	        ELSIF (#i_UDT_PDPStatus.Specific.CircuitBreakerTrippedF108 <> #s_UDT_PDPOldStatus.Specific.CircuitBreakerTrippedF108 AND NOT #sx_SendAllProcedure)
	            OR (#sx_SendAllProcedure AND #ii_ErrorNumber = 10)
	        THEN
	            #sdi_Code := "DB_MFC_ErrorCode".PDP.CircuitBreakerTrippedF108;
	            #si_State := BOOL_TO_INT(#i_UDT_PDPStatus.Specific.CircuitBreakerTrippedF108);
	            #s_UDT_PDPOldStatus.Specific.CircuitBreakerTrippedF108 := #i_UDT_PDPStatus.Specific.CircuitBreakerTrippedF108;
	            #sx_ItemErrorMessageReq := TRUE;
	            #ii_ErrorNumber += 1;
	        ELSIF (#i_UDT_PDPStatus.Specific.CircuitBreakerTrippedF109 <> #s_UDT_PDPOldStatus.Specific.CircuitBreakerTrippedF109 AND NOT #sx_SendAllProcedure)
	            OR (#sx_SendAllProcedure AND #ii_ErrorNumber = 11)
	        THEN
	            #sdi_Code := "DB_MFC_ErrorCode".PDP.CircuitBreakerTrippedF109;
	            #si_State := BOOL_TO_INT(#i_UDT_PDPStatus.Specific.CircuitBreakerTrippedF109);
	            #s_UDT_PDPOldStatus.Specific.CircuitBreakerTrippedF109 := #i_UDT_PDPStatus.Specific.CircuitBreakerTrippedF109;
	            #sx_ItemErrorMessageReq := TRUE;
	            #ii_ErrorNumber += 1;
	        ELSIF (#i_UDT_PDPStatus.Specific.CircuitBreakerTrippedF110 <> #s_UDT_PDPOldStatus.Specific.CircuitBreakerTrippedF110 AND NOT #sx_SendAllProcedure)
	            OR (#sx_SendAllProcedure AND #ii_ErrorNumber = 12)
	        THEN
	            #sdi_Code := "DB_MFC_ErrorCode".PDP.CircuitBreakerTrippedF110;
	            #si_State := BOOL_TO_INT(#i_UDT_PDPStatus.Specific.CircuitBreakerTrippedF110);
	            #s_UDT_PDPOldStatus.Specific.CircuitBreakerTrippedF110 := #i_UDT_PDPStatus.Specific.CircuitBreakerTrippedF110;
	            #sx_ItemErrorMessageReq := TRUE;
	            #ii_ErrorNumber += 1;
	        ELSIF (#i_UDT_PDPStatus.Specific.CircuitBreakerTrippedF111 <> #s_UDT_PDPOldStatus.Specific.CircuitBreakerTrippedF111 AND NOT #sx_SendAllProcedure)
	            OR (#sx_SendAllProcedure AND #ii_ErrorNumber = 13)
	        THEN
	            #sdi_Code := "DB_MFC_ErrorCode".PDP.CircuitBreakerTrippedF111;
	            #si_State := BOOL_TO_INT(#i_UDT_PDPStatus.Specific.CircuitBreakerTrippedF111);
	            #s_UDT_PDPOldStatus.Specific.CircuitBreakerTrippedF111 := #i_UDT_PDPStatus.Specific.CircuitBreakerTrippedF111;
	            #sx_ItemErrorMessageReq := TRUE;
	            #ii_ErrorNumber += 1;
	        ELSIF (#i_UDT_PDPStatus.Specific.CircuitBreakerTrippedF112 <> #s_UDT_PDPOldStatus.Specific.CircuitBreakerTrippedF112 AND NOT #sx_SendAllProcedure)
	            OR (#sx_SendAllProcedure AND #ii_ErrorNumber = 14)
	        THEN
	            #sdi_Code := "DB_MFC_ErrorCode".PDP.CircuitBreakerTrippedF112;
	            #si_State := BOOL_TO_INT(#i_UDT_PDPStatus.Specific.CircuitBreakerTrippedF112);
	            #s_UDT_PDPOldStatus.Specific.CircuitBreakerTrippedF112 := #i_UDT_PDPStatus.Specific.CircuitBreakerTrippedF112;
	            #sx_ItemErrorMessageReq := TRUE;
	            #ii_ErrorNumber += 1;
	        ELSIF (#i_UDT_PDPStatus.Specific.CircuitBreakerTrippedF113 <> #s_UDT_PDPOldStatus.Specific.CircuitBreakerTrippedF113 AND NOT #sx_SendAllProcedure)
	            OR (#sx_SendAllProcedure AND #ii_ErrorNumber = 15)
	        THEN
	            #sdi_Code := "DB_MFC_ErrorCode".PDP.CircuitBreakerTrippedF113;
	            #si_State := BOOL_TO_INT(#i_UDT_PDPStatus.Specific.CircuitBreakerTrippedF113);
	            #s_UDT_PDPOldStatus.Specific.CircuitBreakerTrippedF113 := #i_UDT_PDPStatus.Specific.CircuitBreakerTrippedF113;
	            #sx_ItemErrorMessageReq := TRUE;
	            #ii_ErrorNumber += 1;
	        ELSIF (#i_UDT_PDPStatus.Specific.CircuitBreakerTrippedF114 <> #s_UDT_PDPOldStatus.Specific.CircuitBreakerTrippedF114 AND NOT #sx_SendAllProcedure)
	            OR (#sx_SendAllProcedure AND #ii_ErrorNumber = 16)
	        THEN
	            #sdi_Code := "DB_MFC_ErrorCode".PDP.CircuitBreakerTrippedF114;
	            #si_State := BOOL_TO_INT(#i_UDT_PDPStatus.Specific.CircuitBreakerTrippedF114);
	            #s_UDT_PDPOldStatus.Specific.CircuitBreakerTrippedF114 := #i_UDT_PDPStatus.Specific.CircuitBreakerTrippedF114;
	            #sx_ItemErrorMessageReq := TRUE;
	            #ii_ErrorNumber += 1;
	        ELSIF (#i_UDT_PDPStatus.Specific.CircuitBreakerTrippedF115 <> #s_UDT_PDPOldStatus.Specific.CircuitBreakerTrippedF115 AND NOT #sx_SendAllProcedure)
	            OR (#sx_SendAllProcedure AND #ii_ErrorNumber = 17)
	        THEN
	            #sdi_Code := "DB_MFC_ErrorCode".PDP.CircuitBreakerTrippedF115;
	            #si_State := BOOL_TO_INT(#i_UDT_PDPStatus.Specific.CircuitBreakerTrippedF115);
	            #s_UDT_PDPOldStatus.Specific.CircuitBreakerTrippedF115 := #i_UDT_PDPStatus.Specific.CircuitBreakerTrippedF115;
	            #sx_ItemErrorMessageReq := TRUE;
	            #ii_ErrorNumber += 1;
	        ELSIF (#i_UDT_PDPStatus.Specific.CircuitBreakerTrippedF116 <> #s_UDT_PDPOldStatus.Specific.CircuitBreakerTrippedF116 AND NOT #sx_SendAllProcedure)
	            OR (#sx_SendAllProcedure AND #ii_ErrorNumber = 18)
	        THEN
	            #sdi_Code := "DB_MFC_ErrorCode".PDP.CircuitBreakerTrippedF116;
	            #si_State := BOOL_TO_INT(#i_UDT_PDPStatus.Specific.CircuitBreakerTrippedF116);
	            #s_UDT_PDPOldStatus.Specific.CircuitBreakerTrippedF116 := #i_UDT_PDPStatus.Specific.CircuitBreakerTrippedF116;
	            #sx_ItemErrorMessageReq := TRUE;
	            #ii_ErrorNumber += 1;
	        ELSIF (#i_UDT_PDPStatus.Specific.CircuitBreakerTrippedF117 <> #s_UDT_PDPOldStatus.Specific.CircuitBreakerTrippedF117 AND NOT #sx_SendAllProcedure)
	            OR (#sx_SendAllProcedure AND #ii_ErrorNumber = 19)
	        THEN
	            #sdi_Code := "DB_MFC_ErrorCode".PDP.CircuitBreakerTrippedF117;
	            #si_State := BOOL_TO_INT(#i_UDT_PDPStatus.Specific.CircuitBreakerTrippedF117);
	            #s_UDT_PDPOldStatus.Specific.CircuitBreakerTrippedF117 := #i_UDT_PDPStatus.Specific.CircuitBreakerTrippedF117;
	            #sx_ItemErrorMessageReq := TRUE;
	            #ii_ErrorNumber += 1;
	        ELSIF (#i_UDT_PDPStatus.Specific.CircuitBreakerTrippedF118 <> #s_UDT_PDPOldStatus.Specific.CircuitBreakerTrippedF118 AND NOT #sx_SendAllProcedure)
	            OR (#sx_SendAllProcedure AND #ii_ErrorNumber = 20)
	        THEN
	            #sdi_Code := "DB_MFC_ErrorCode".PDP.CircuitBreakerTrippedF118;
	            #si_State := BOOL_TO_INT(#i_UDT_PDPStatus.Specific.CircuitBreakerTrippedF118);
	            #s_UDT_PDPOldStatus.Specific.CircuitBreakerTrippedF118 := #i_UDT_PDPStatus.Specific.CircuitBreakerTrippedF118;
	            #sx_ItemErrorMessageReq := TRUE;
	            #ii_ErrorNumber += 1;
	        ELSIF (#i_UDT_PDPStatus.Specific.CircuitBreakerTrippedF119 <> #s_UDT_PDPOldStatus.Specific.CircuitBreakerTrippedF119 AND NOT #sx_SendAllProcedure)
	            OR (#sx_SendAllProcedure AND #ii_ErrorNumber = 21)
	        THEN
	            #sdi_Code := "DB_MFC_ErrorCode".PDP.CircuitBreakerTrippedF119;
	            #si_State := BOOL_TO_INT(#i_UDT_PDPStatus.Specific.CircuitBreakerTrippedF119);
	            #s_UDT_PDPOldStatus.Specific.CircuitBreakerTrippedF119 := #i_UDT_PDPStatus.Specific.CircuitBreakerTrippedF119;
	            #sx_ItemErrorMessageReq := TRUE;
	            #ii_ErrorNumber += 1;
	        ELSIF (#i_UDT_PDPStatus.Specific.CircuitBreakerTrippedF120 <> #s_UDT_PDPOldStatus.Specific.CircuitBreakerTrippedF120 AND NOT #sx_SendAllProcedure)
	            OR (#sx_SendAllProcedure AND #ii_ErrorNumber = 22)
	        THEN
	            #sdi_Code := "DB_MFC_ErrorCode".PDP.CircuitBreakerTrippedF120;
	            #si_State := BOOL_TO_INT(#i_UDT_PDPStatus.Specific.CircuitBreakerTrippedF120);
	            #s_UDT_PDPOldStatus.Specific.CircuitBreakerTrippedF120 := #i_UDT_PDPStatus.Specific.CircuitBreakerTrippedF120;
	            #sx_ItemErrorMessageReq := TRUE;
	            #ii_ErrorNumber += 1;
	        ELSIF (#i_UDT_PDPStatus.Specific.CircuitBreakerTrippedF121 <> #s_UDT_PDPOldStatus.Specific.CircuitBreakerTrippedF121 AND NOT #sx_SendAllProcedure)
	            OR (#sx_SendAllProcedure AND #ii_ErrorNumber = 23)
	        THEN
	            #sdi_Code := "DB_MFC_ErrorCode".PDP.CircuitBreakerTrippedF121;
	            #si_State := BOOL_TO_INT(#i_UDT_PDPStatus.Specific.CircuitBreakerTrippedF121);
	            #s_UDT_PDPOldStatus.Specific.CircuitBreakerTrippedF121 := #i_UDT_PDPStatus.Specific.CircuitBreakerTrippedF121;
	            #sx_ItemErrorMessageReq := TRUE;
	            #ii_ErrorNumber += 1;
	        ELSIF (#i_UDT_PDPStatus.Specific.CircuitBreakerTrippedF122 <> #s_UDT_PDPOldStatus.Specific.CircuitBreakerTrippedF122 AND NOT #sx_SendAllProcedure)
	            OR (#sx_SendAllProcedure AND #ii_ErrorNumber = 24)
	        THEN
	            #sdi_Code := "DB_MFC_ErrorCode".PDP.CircuitBreakerTrippedF122;
	            #si_State := BOOL_TO_INT(#i_UDT_PDPStatus.Specific.CircuitBreakerTrippedF122);
	            #s_UDT_PDPOldStatus.Specific.CircuitBreakerTrippedF122 := #i_UDT_PDPStatus.Specific.CircuitBreakerTrippedF122;
	            #sx_ItemErrorMessageReq := TRUE;
	            #ii_ErrorNumber += 1;
	        ELSIF (#i_UDT_PDPStatus.Specific.CircuitBreakerTrippedF123 <> #s_UDT_PDPOldStatus.Specific.CircuitBreakerTrippedF123 AND NOT #sx_SendAllProcedure)
	            OR (#sx_SendAllProcedure AND #ii_ErrorNumber = 25)
	        THEN
	            #sdi_Code := "DB_MFC_ErrorCode".PDP.CircuitBreakerTrippedF123;
	            #si_State := BOOL_TO_INT(#i_UDT_PDPStatus.Specific.CircuitBreakerTrippedF123);
	            #s_UDT_PDPOldStatus.Specific.CircuitBreakerTrippedF123 := #i_UDT_PDPStatus.Specific.CircuitBreakerTrippedF123;
	            #sx_ItemErrorMessageReq := TRUE;
	            #ii_ErrorNumber += 1;
	        ELSIF (#i_UDT_PDPStatus.Specific.CircuitBreakerTrippedF124 <> #s_UDT_PDPOldStatus.Specific.CircuitBreakerTrippedF124 AND NOT #sx_SendAllProcedure)
	            OR (#sx_SendAllProcedure AND #ii_ErrorNumber = 26)
	        THEN
	            #sdi_Code := "DB_MFC_ErrorCode".PDP.CircuitBreakerTrippedF124;
	            #si_State := BOOL_TO_INT(#i_UDT_PDPStatus.Specific.CircuitBreakerTrippedF124);
	            #s_UDT_PDPOldStatus.Specific.CircuitBreakerTrippedF124 := #i_UDT_PDPStatus.Specific.CircuitBreakerTrippedF124;
	            #sx_ItemErrorMessageReq := TRUE;
	            #ii_ErrorNumber += 1;
	        ELSIF (#i_UDT_PDPStatus.Specific.CircuitBreakerTrippedF125 <> #s_UDT_PDPOldStatus.Specific.CircuitBreakerTrippedF125 AND NOT #sx_SendAllProcedure)
	            OR (#sx_SendAllProcedure AND #ii_ErrorNumber = 27)
	        THEN
	            #sdi_Code := "DB_MFC_ErrorCode".PDP.CircuitBreakerTrippedF125;
	            #si_State := BOOL_TO_INT(#i_UDT_PDPStatus.Specific.CircuitBreakerTrippedF125);
	            #s_UDT_PDPOldStatus.Specific.CircuitBreakerTrippedF125 := #i_UDT_PDPStatus.Specific.CircuitBreakerTrippedF125;
	            #sx_ItemErrorMessageReq := TRUE;
	            #ii_ErrorNumber += 1;
	        ELSIF (#i_UDT_PDPStatus.Specific.CircuitBreakerTrippedF126 <> #s_UDT_PDPOldStatus.Specific.CircuitBreakerTrippedF126 AND NOT #sx_SendAllProcedure)
	            OR (#sx_SendAllProcedure AND #ii_ErrorNumber = 28)
	        THEN
	            #sdi_Code := "DB_MFC_ErrorCode".PDP.CircuitBreakerTrippedF126;
	            #si_State := BOOL_TO_INT(#i_UDT_PDPStatus.Specific.CircuitBreakerTrippedF126);
	            #s_UDT_PDPOldStatus.Specific.CircuitBreakerTrippedF126 := #i_UDT_PDPStatus.Specific.CircuitBreakerTrippedF126;
	            #sx_ItemErrorMessageReq := TRUE;
	            #ii_ErrorNumber += 1;
	        ELSIF (#i_UDT_PDPStatus.Specific.CircuitBreakerTrippedF127 <> #s_UDT_PDPOldStatus.Specific.CircuitBreakerTrippedF127 AND NOT #sx_SendAllProcedure)
	            OR (#sx_SendAllProcedure AND #ii_ErrorNumber = 29)
	        THEN
	            #sdi_Code := "DB_MFC_ErrorCode".PDP.CircuitBreakerTrippedF127;
	            #si_State := BOOL_TO_INT(#i_UDT_PDPStatus.Specific.CircuitBreakerTrippedF127);
	            #s_UDT_PDPOldStatus.Specific.CircuitBreakerTrippedF127 := #i_UDT_PDPStatus.Specific.CircuitBreakerTrippedF127;
	            #sx_ItemErrorMessageReq := TRUE;
	            #ii_ErrorNumber += 1;
	        ELSIF (#i_UDT_PDPStatus.Specific.CircuitBreakerTrippedF128 <> #s_UDT_PDPOldStatus.Specific.CircuitBreakerTrippedF128 AND NOT #sx_SendAllProcedure)
	            OR (#sx_SendAllProcedure AND #ii_ErrorNumber = 30)
	        THEN
	            #sdi_Code := "DB_MFC_ErrorCode".PDP.CircuitBreakerTrippedF128;
	            #si_State := BOOL_TO_INT(#i_UDT_PDPStatus.Specific.CircuitBreakerTrippedF128);
	            #s_UDT_PDPOldStatus.Specific.CircuitBreakerTrippedF128 := #i_UDT_PDPStatus.Specific.CircuitBreakerTrippedF128;
	            #sx_ItemErrorMessageReq := TRUE;
	            #ii_ErrorNumber += 1;
	        ELSIF (#i_UDT_PDPStatus.Specific.CircuitBreakerTrippedF129 <> #s_UDT_PDPOldStatus.Specific.CircuitBreakerTrippedF129 AND NOT #sx_SendAllProcedure)
	            OR (#sx_SendAllProcedure AND #ii_ErrorNumber = 31)
	        THEN
	            #sdi_Code := "DB_MFC_ErrorCode".PDP.CircuitBreakerTrippedF129;
	            #si_State := BOOL_TO_INT(#i_UDT_PDPStatus.Specific.CircuitBreakerTrippedF129);
	            #s_UDT_PDPOldStatus.Specific.CircuitBreakerTrippedF129 := #i_UDT_PDPStatus.Specific.CircuitBreakerTrippedF129;
	            #sx_ItemErrorMessageReq := TRUE;
	            #ii_ErrorNumber += 1;
	        ELSIF (#i_UDT_PDPStatus.Specific.CircuitBreakerTrippedF130 <> #s_UDT_PDPOldStatus.Specific.CircuitBreakerTrippedF130 AND NOT #sx_SendAllProcedure)
	            OR (#sx_SendAllProcedure AND #ii_ErrorNumber = 32)
	        THEN
	            #sdi_Code := "DB_MFC_ErrorCode".PDP.CircuitBreakerTrippedF130;
	            #si_State := BOOL_TO_INT(#i_UDT_PDPStatus.Specific.CircuitBreakerTrippedF130);
	            #s_UDT_PDPOldStatus.Specific.CircuitBreakerTrippedF130 := #i_UDT_PDPStatus.Specific.CircuitBreakerTrippedF130;
	            #sx_ItemErrorMessageReq := TRUE;
	            #ii_ErrorNumber += 1;
	        ELSIF (#i_UDT_PDPStatus.Specific.CircuitBreakerTrippedF131 <> #s_UDT_PDPOldStatus.Specific.CircuitBreakerTrippedF131 AND NOT #sx_SendAllProcedure)
	            OR (#sx_SendAllProcedure AND #ii_ErrorNumber = 33)
	        THEN
	            #sdi_Code := "DB_MFC_ErrorCode".PDP.CircuitBreakerTrippedF131;
	            #si_State := BOOL_TO_INT(#i_UDT_PDPStatus.Specific.CircuitBreakerTrippedF131);
	            #s_UDT_PDPOldStatus.Specific.CircuitBreakerTrippedF131 := #i_UDT_PDPStatus.Specific.CircuitBreakerTrippedF131;
	            #sx_ItemErrorMessageReq := TRUE;
	            #ii_ErrorNumber += 1;
	        ELSIF (#i_UDT_PDPStatus.Specific.CircuitBreakerTrippedF132 <> #s_UDT_PDPOldStatus.Specific.CircuitBreakerTrippedF132 AND NOT #sx_SendAllProcedure)
	            OR (#sx_SendAllProcedure AND #ii_ErrorNumber = 34)
	        THEN
	            #sdi_Code := "DB_MFC_ErrorCode".PDP.CircuitBreakerTrippedF132;
	            #si_State := BOOL_TO_INT(#i_UDT_PDPStatus.Specific.CircuitBreakerTrippedF132);
	            #s_UDT_PDPOldStatus.Specific.CircuitBreakerTrippedF132 := #i_UDT_PDPStatus.Specific.CircuitBreakerTrippedF132;
	            #sx_ItemErrorMessageReq := TRUE;
	            #ii_ErrorNumber += 1;
	        ELSIF (#i_UDT_PDPStatus.Specific.CircuitBreakerTrippedF133 <> #s_UDT_PDPOldStatus.Specific.CircuitBreakerTrippedF133 AND NOT #sx_SendAllProcedure)
	            OR (#sx_SendAllProcedure AND #ii_ErrorNumber = 35)
	        THEN
	            #sdi_Code := "DB_MFC_ErrorCode".PDP.CircuitBreakerTrippedF133;
	            #si_State := BOOL_TO_INT(#i_UDT_PDPStatus.Specific.CircuitBreakerTrippedF133);
	            #s_UDT_PDPOldStatus.Specific.CircuitBreakerTrippedF133 := #i_UDT_PDPStatus.Specific.CircuitBreakerTrippedF133;
	            #sx_ItemErrorMessageReq := TRUE;
	            #ii_ErrorNumber += 1;
	        ELSIF (#i_UDT_PDPStatus.Specific.CircuitBreakerTrippedF134 <> #s_UDT_PDPOldStatus.Specific.CircuitBreakerTrippedF134 AND NOT #sx_SendAllProcedure)
	            OR (#sx_SendAllProcedure AND #ii_ErrorNumber = 36)
	        THEN
	            #sdi_Code := "DB_MFC_ErrorCode".PDP.CircuitBreakerTrippedF134;
	            #si_State := BOOL_TO_INT(#i_UDT_PDPStatus.Specific.CircuitBreakerTrippedF134);
	            #s_UDT_PDPOldStatus.Specific.CircuitBreakerTrippedF134 := #i_UDT_PDPStatus.Specific.CircuitBreakerTrippedF134;
	            #sx_ItemErrorMessageReq := TRUE;
	            #ii_ErrorNumber += 1;
	        ELSIF (#i_UDT_PDPStatus.Specific.CircuitBreakerTrippedF135 <> #s_UDT_PDPOldStatus.Specific.CircuitBreakerTrippedF135 AND NOT #sx_SendAllProcedure)
	            OR (#sx_SendAllProcedure AND #ii_ErrorNumber = 37)
	        THEN
	            #sdi_Code := "DB_MFC_ErrorCode".PDP.CircuitBreakerTrippedF135;
	            #si_State := BOOL_TO_INT(#i_UDT_PDPStatus.Specific.CircuitBreakerTrippedF135);
	            #s_UDT_PDPOldStatus.Specific.CircuitBreakerTrippedF135 := #i_UDT_PDPStatus.Specific.CircuitBreakerTrippedF135;
	            #sx_ItemErrorMessageReq := TRUE;
	            #ii_ErrorNumber += 1;
	        ELSIF (#i_UDT_PDPStatus.Specific.CircuitBreakerTrippedF201 <> #s_UDT_PDPOldStatus.Specific.CircuitBreakerTrippedF201 AND NOT #sx_SendAllProcedure)
	            OR (#sx_SendAllProcedure AND #ii_ErrorNumber = 38)
	        THEN
	            #sdi_Code := "DB_MFC_ErrorCode".PDP.CircuitBreakerTrippedF201;
	            #si_State := BOOL_TO_INT(#i_UDT_PDPStatus.Specific.CircuitBreakerTrippedF201);
	            #s_UDT_PDPOldStatus.Specific.CircuitBreakerTrippedF201 := #i_UDT_PDPStatus.Specific.CircuitBreakerTrippedF201;
	            #sx_ItemErrorMessageReq := TRUE;
	            #ii_ErrorNumber += 1;
	        ELSIF (#i_UDT_PDPStatus.Specific.CircuitBreakerTrippedF202 <> #s_UDT_PDPOldStatus.Specific.CircuitBreakerTrippedF202 AND NOT #sx_SendAllProcedure)
	            OR (#sx_SendAllProcedure AND #ii_ErrorNumber = 39)
	        THEN
	            #sdi_Code := "DB_MFC_ErrorCode".PDP.CircuitBreakerTrippedF202;
	            #si_State := BOOL_TO_INT(#i_UDT_PDPStatus.Specific.CircuitBreakerTrippedF202);
	            #s_UDT_PDPOldStatus.Specific.CircuitBreakerTrippedF202 := #i_UDT_PDPStatus.Specific.CircuitBreakerTrippedF202;
	            #sx_ItemErrorMessageReq := TRUE;
	            #ii_ErrorNumber += 1;
	        ELSIF (#i_UDT_PDPStatus.Specific.CircuitBreakerTrippedF203 <> #s_UDT_PDPOldStatus.Specific.CircuitBreakerTrippedF203 AND NOT #sx_SendAllProcedure)
	            OR (#sx_SendAllProcedure AND #ii_ErrorNumber = 40)
	        THEN
	            #sdi_Code := "DB_MFC_ErrorCode".PDP.CircuitBreakerTrippedF203;
	            #si_State := BOOL_TO_INT(#i_UDT_PDPStatus.Specific.CircuitBreakerTrippedF203);
	            #s_UDT_PDPOldStatus.Specific.CircuitBreakerTrippedF203 := #i_UDT_PDPStatus.Specific.CircuitBreakerTrippedF203;
	            #sx_ItemErrorMessageReq := TRUE;
	            #ii_ErrorNumber += 1;
	        ELSIF (#i_UDT_PDPStatus.Specific.CircuitBreakerTrippedF204 <> #s_UDT_PDPOldStatus.Specific.CircuitBreakerTrippedF204 AND NOT #sx_SendAllProcedure)
	            OR (#sx_SendAllProcedure AND #ii_ErrorNumber = 41)
	        THEN
	            #sdi_Code := "DB_MFC_ErrorCode".PDP.CircuitBreakerTrippedF204;
	            #si_State := BOOL_TO_INT(#i_UDT_PDPStatus.Specific.CircuitBreakerTrippedF204);
	            #s_UDT_PDPOldStatus.Specific.CircuitBreakerTrippedF204 := #i_UDT_PDPStatus.Specific.CircuitBreakerTrippedF204;
	            #sx_ItemErrorMessageReq := TRUE;
	            #ii_ErrorNumber += 1;
	        ELSIF (#i_UDT_PDPStatus.Specific.CircuitBreakerTrippedF205 <> #s_UDT_PDPOldStatus.Specific.CircuitBreakerTrippedF205 AND NOT #sx_SendAllProcedure)
	            OR (#sx_SendAllProcedure AND #ii_ErrorNumber = 42)
	        THEN
	            #sdi_Code := "DB_MFC_ErrorCode".PDP.CircuitBreakerTrippedF205;
	            #si_State := BOOL_TO_INT(#i_UDT_PDPStatus.Specific.CircuitBreakerTrippedF205);
	            #s_UDT_PDPOldStatus.Specific.CircuitBreakerTrippedF205 := #i_UDT_PDPStatus.Specific.CircuitBreakerTrippedF205;
	            #sx_ItemErrorMessageReq := TRUE;
	            #ii_ErrorNumber += 1;
	        ELSIF (#i_UDT_PDPStatus.Specific.CircuitBreakerTrippedF206 <> #s_UDT_PDPOldStatus.Specific.CircuitBreakerTrippedF206 AND NOT #sx_SendAllProcedure)
	            OR (#sx_SendAllProcedure AND #ii_ErrorNumber = 43)
	        THEN
	            #sdi_Code := "DB_MFC_ErrorCode".PDP.CircuitBreakerTrippedF206;
	            #si_State := BOOL_TO_INT(#i_UDT_PDPStatus.Specific.CircuitBreakerTrippedF206);
	            #s_UDT_PDPOldStatus.Specific.CircuitBreakerTrippedF206 := #i_UDT_PDPStatus.Specific.CircuitBreakerTrippedF206;
	            #sx_ItemErrorMessageReq := TRUE;
	            #ii_ErrorNumber += 1;
	        ELSIF (#i_UDT_PDPStatus.Specific.CircuitBreakerTrippedF207 <> #s_UDT_PDPOldStatus.Specific.CircuitBreakerTrippedF207 AND NOT #sx_SendAllProcedure)
	            OR (#sx_SendAllProcedure AND #ii_ErrorNumber = 44)
	        THEN
	            #sdi_Code := "DB_MFC_ErrorCode".PDP.CircuitBreakerTrippedF207;
	            #si_State := BOOL_TO_INT(#i_UDT_PDPStatus.Specific.CircuitBreakerTrippedF207);
	            #s_UDT_PDPOldStatus.Specific.CircuitBreakerTrippedF207 := #i_UDT_PDPStatus.Specific.CircuitBreakerTrippedF207;
	            #sx_ItemErrorMessageReq := TRUE;
	            #ii_ErrorNumber += 1;
	        ELSIF (#i_UDT_PDPStatus.Specific.CircuitBreakerTrippedF208 <> #s_UDT_PDPOldStatus.Specific.CircuitBreakerTrippedF208 AND NOT #sx_SendAllProcedure)
	            OR (#sx_SendAllProcedure AND #ii_ErrorNumber = 45)
	        THEN
	            #sdi_Code := "DB_MFC_ErrorCode".PDP.CircuitBreakerTrippedF208;
	            #si_State := BOOL_TO_INT(#i_UDT_PDPStatus.Specific.CircuitBreakerTrippedF208);
	            #s_UDT_PDPOldStatus.Specific.CircuitBreakerTrippedF208 := #i_UDT_PDPStatus.Specific.CircuitBreakerTrippedF208;
	            #sx_ItemErrorMessageReq := TRUE;
	            #ii_ErrorNumber += 1;
	        ELSIF (#i_UDT_PDPStatus.Specific.CircuitBreakerTrippedF209 <> #s_UDT_PDPOldStatus.Specific.CircuitBreakerTrippedF209 AND NOT #sx_SendAllProcedure)
	            OR (#sx_SendAllProcedure AND #ii_ErrorNumber = 46)
	        THEN
	            #sdi_Code := "DB_MFC_ErrorCode".PDP.CircuitBreakerTrippedF209;
	            #si_State := BOOL_TO_INT(#i_UDT_PDPStatus.Specific.CircuitBreakerTrippedF209);
	            #s_UDT_PDPOldStatus.Specific.CircuitBreakerTrippedF209 := #i_UDT_PDPStatus.Specific.CircuitBreakerTrippedF209;
	            #sx_ItemErrorMessageReq := TRUE;
	            #ii_ErrorNumber += 1;
	        ELSIF (#i_UDT_PDPStatus.Specific.CircuitBreakerTrippedF210 <> #s_UDT_PDPOldStatus.Specific.CircuitBreakerTrippedF210 AND NOT #sx_SendAllProcedure)
	            OR (#sx_SendAllProcedure AND #ii_ErrorNumber = 47)
	        THEN
	            #sdi_Code := "DB_MFC_ErrorCode".PDP.CircuitBreakerTrippedF210;
	            #si_State := BOOL_TO_INT(#i_UDT_PDPStatus.Specific.CircuitBreakerTrippedF210);
	            #s_UDT_PDPOldStatus.Specific.CircuitBreakerTrippedF210 := #i_UDT_PDPStatus.Specific.CircuitBreakerTrippedF210;
	            #sx_ItemErrorMessageReq := TRUE;
	            #ii_ErrorNumber += 1;
	        ELSIF (#i_UDT_PDPStatus.Specific.CircuitBreakerTrippedF211 <> #s_UDT_PDPOldStatus.Specific.CircuitBreakerTrippedF211 AND NOT #sx_SendAllProcedure)
	            OR (#sx_SendAllProcedure AND #ii_ErrorNumber = 48)
	        THEN
	            #sdi_Code := "DB_MFC_ErrorCode".PDP.CircuitBreakerTrippedF211;
	            #si_State := BOOL_TO_INT(#i_UDT_PDPStatus.Specific.CircuitBreakerTrippedF211);
	            #s_UDT_PDPOldStatus.Specific.CircuitBreakerTrippedF211 := #i_UDT_PDPStatus.Specific.CircuitBreakerTrippedF211;
	            #sx_ItemErrorMessageReq := TRUE;
	            #ii_ErrorNumber += 1;
	        ELSIF (#i_UDT_PDPStatus.Specific.CircuitBreakerTrippedF212 <> #s_UDT_PDPOldStatus.Specific.CircuitBreakerTrippedF212 AND NOT #sx_SendAllProcedure)
	            OR (#sx_SendAllProcedure AND #ii_ErrorNumber = 49)
	        THEN
	            #sdi_Code := "DB_MFC_ErrorCode".PDP.CircuitBreakerTrippedF212;
	            #si_State := BOOL_TO_INT(#i_UDT_PDPStatus.Specific.CircuitBreakerTrippedF212);
	            #s_UDT_PDPOldStatus.Specific.CircuitBreakerTrippedF212 := #i_UDT_PDPStatus.Specific.CircuitBreakerTrippedF212;
	            #sx_ItemErrorMessageReq := TRUE;
	            #ii_ErrorNumber += 1;
	        ELSIF (#i_UDT_PDPStatus.Specific.CircuitBreakerTrippedF213 <> #s_UDT_PDPOldStatus.Specific.CircuitBreakerTrippedF213 AND NOT #sx_SendAllProcedure)
	            OR (#sx_SendAllProcedure AND #ii_ErrorNumber = 50)
	        THEN
	            #sdi_Code := "DB_MFC_ErrorCode".PDP.CircuitBreakerTrippedF213;
	            #si_State := BOOL_TO_INT(#i_UDT_PDPStatus.Specific.CircuitBreakerTrippedF213);
	            #s_UDT_PDPOldStatus.Specific.CircuitBreakerTrippedF213 := #i_UDT_PDPStatus.Specific.CircuitBreakerTrippedF213;
	            #sx_ItemErrorMessageReq := TRUE;
	            #ii_ErrorNumber += 1;
	        ELSIF (#i_UDT_PDPStatus.Specific.CircuitBreakerTrippedF214 <> #s_UDT_PDPOldStatus.Specific.CircuitBreakerTrippedF214 AND NOT #sx_SendAllProcedure)
	            OR (#sx_SendAllProcedure AND #ii_ErrorNumber = 51)
	        THEN
	            #sdi_Code := "DB_MFC_ErrorCode".PDP.CircuitBreakerTrippedF214;
	            #si_State := BOOL_TO_INT(#i_UDT_PDPStatus.Specific.CircuitBreakerTrippedF214);
	            #s_UDT_PDPOldStatus.Specific.CircuitBreakerTrippedF214 := #i_UDT_PDPStatus.Specific.CircuitBreakerTrippedF214;
	            #sx_ItemErrorMessageReq := TRUE;
	            #ii_ErrorNumber += 1;
	        ELSIF (#i_UDT_PDPStatus.Specific.CircuitBreakerTrippedF215 <> #s_UDT_PDPOldStatus.Specific.CircuitBreakerTrippedF215 AND NOT #sx_SendAllProcedure)
	            OR (#sx_SendAllProcedure AND #ii_ErrorNumber = 52)
	        THEN
	            #sdi_Code := "DB_MFC_ErrorCode".PDP.CircuitBreakerTrippedF215;
	            #si_State := BOOL_TO_INT(#i_UDT_PDPStatus.Specific.CircuitBreakerTrippedF215);
	            #s_UDT_PDPOldStatus.Specific.CircuitBreakerTrippedF215 := #i_UDT_PDPStatus.Specific.CircuitBreakerTrippedF215;
	            #sx_ItemErrorMessageReq := TRUE;
	            #ii_ErrorNumber += 1;
	        ELSIF (#i_UDT_PDPStatus.Specific.CircuitBreakerTrippedF216 <> #s_UDT_PDPOldStatus.Specific.CircuitBreakerTrippedF216 AND NOT #sx_SendAllProcedure)
	            OR (#sx_SendAllProcedure AND #ii_ErrorNumber = 53)
	        THEN
	            #sdi_Code := "DB_MFC_ErrorCode".PDP.CircuitBreakerTrippedF216;
	            #si_State := BOOL_TO_INT(#i_UDT_PDPStatus.Specific.CircuitBreakerTrippedF216);
	            #s_UDT_PDPOldStatus.Specific.CircuitBreakerTrippedF216 := #i_UDT_PDPStatus.Specific.CircuitBreakerTrippedF216;
	            #sx_ItemErrorMessageReq := TRUE;
	            #ii_ErrorNumber += 1;
	        ELSIF (#i_UDT_PDPStatus.Specific.CircuitBreakerTrippedF217 <> #s_UDT_PDPOldStatus.Specific.CircuitBreakerTrippedF217 AND NOT #sx_SendAllProcedure)
	            OR (#sx_SendAllProcedure AND #ii_ErrorNumber = 54)
	        THEN
	            #sdi_Code := "DB_MFC_ErrorCode".PDP.CircuitBreakerTrippedF217;
	            #si_State := BOOL_TO_INT(#i_UDT_PDPStatus.Specific.CircuitBreakerTrippedF217);
	            #s_UDT_PDPOldStatus.Specific.CircuitBreakerTrippedF217 := #i_UDT_PDPStatus.Specific.CircuitBreakerTrippedF217;
	            #sx_ItemErrorMessageReq := TRUE;
	            #ii_ErrorNumber += 1;
	        ELSIF (#i_UDT_PDPStatus.Specific.CircuitBreakerTrippedF218 <> #s_UDT_PDPOldStatus.Specific.CircuitBreakerTrippedF218 AND NOT #sx_SendAllProcedure)
	            OR (#sx_SendAllProcedure AND #ii_ErrorNumber = 55)
	        THEN
	            #sdi_Code := "DB_MFC_ErrorCode".PDP.CircuitBreakerTrippedF218;
	            #si_State := BOOL_TO_INT(#i_UDT_PDPStatus.Specific.CircuitBreakerTrippedF218);
	            #s_UDT_PDPOldStatus.Specific.CircuitBreakerTrippedF218 := #i_UDT_PDPStatus.Specific.CircuitBreakerTrippedF218;
	            #sx_ItemErrorMessageReq := TRUE;
	            #ii_ErrorNumber += 1;
	        ELSIF (#i_UDT_PDPStatus.Specific.CircuitBreakerTrippedF219 <> #s_UDT_PDPOldStatus.Specific.CircuitBreakerTrippedF219 AND NOT #sx_SendAllProcedure)
	            OR (#sx_SendAllProcedure AND #ii_ErrorNumber = 56)
	        THEN
	            #sdi_Code := "DB_MFC_ErrorCode".PDP.CircuitBreakerTrippedF219;
	            #si_State := BOOL_TO_INT(#i_UDT_PDPStatus.Specific.CircuitBreakerTrippedF219);
	            #s_UDT_PDPOldStatus.Specific.CircuitBreakerTrippedF219 := #i_UDT_PDPStatus.Specific.CircuitBreakerTrippedF219;
	            #sx_ItemErrorMessageReq := TRUE;
	            #ii_ErrorNumber += 1;
	        ELSIF (#i_UDT_PDPStatus.Specific.CircuitBreakerTrippedF220 <> #s_UDT_PDPOldStatus.Specific.CircuitBreakerTrippedF220 AND NOT #sx_SendAllProcedure)
	            OR (#sx_SendAllProcedure AND #ii_ErrorNumber = 57)
	        THEN
	            #sdi_Code := "DB_MFC_ErrorCode".PDP.CircuitBreakerTrippedF220;
	            #si_State := BOOL_TO_INT(#i_UDT_PDPStatus.Specific.CircuitBreakerTrippedF220);
	            #s_UDT_PDPOldStatus.Specific.CircuitBreakerTrippedF220 := #i_UDT_PDPStatus.Specific.CircuitBreakerTrippedF220;
	            #sx_ItemErrorMessageReq := TRUE;
	            #ii_ErrorNumber += 1;
	        ELSIF (#i_UDT_PDPStatus.Specific.CircuitBreakerTrippedF221 <> #s_UDT_PDPOldStatus.Specific.CircuitBreakerTrippedF221 AND NOT #sx_SendAllProcedure)
	            OR (#sx_SendAllProcedure AND #ii_ErrorNumber = 58)
	        THEN
	            #sdi_Code := "DB_MFC_ErrorCode".PDP.CircuitBreakerTrippedF221;
	            #si_State := BOOL_TO_INT(#i_UDT_PDPStatus.Specific.CircuitBreakerTrippedF221);
	            #s_UDT_PDPOldStatus.Specific.CircuitBreakerTrippedF221 := #i_UDT_PDPStatus.Specific.CircuitBreakerTrippedF221;
	            #sx_ItemErrorMessageReq := TRUE;
	            #ii_ErrorNumber += 1;
	        ELSIF (#i_UDT_PDPStatus.Specific.CircuitBreakerTrippedF222 <> #s_UDT_PDPOldStatus.Specific.CircuitBreakerTrippedF222 AND NOT #sx_SendAllProcedure)
	            OR (#sx_SendAllProcedure AND #ii_ErrorNumber = 59)
	        THEN
	            #sdi_Code := "DB_MFC_ErrorCode".PDP.CircuitBreakerTrippedF222;
	            #si_State := BOOL_TO_INT(#i_UDT_PDPStatus.Specific.CircuitBreakerTrippedF222);
	            #s_UDT_PDPOldStatus.Specific.CircuitBreakerTrippedF222 := #i_UDT_PDPStatus.Specific.CircuitBreakerTrippedF222;
	            #sx_ItemErrorMessageReq := TRUE;
	            #ii_ErrorNumber += 1;
	        ELSIF (#i_UDT_PDPStatus.Specific.CircuitBreakerTrippedF223 <> #s_UDT_PDPOldStatus.Specific.CircuitBreakerTrippedF223 AND NOT #sx_SendAllProcedure)
	            OR (#sx_SendAllProcedure AND #ii_ErrorNumber = 60)
	        THEN
	            #sdi_Code := "DB_MFC_ErrorCode".PDP.CircuitBreakerTrippedF223;
	            #si_State := BOOL_TO_INT(#i_UDT_PDPStatus.Specific.CircuitBreakerTrippedF223);
	            #s_UDT_PDPOldStatus.Specific.CircuitBreakerTrippedF223 := #i_UDT_PDPStatus.Specific.CircuitBreakerTrippedF223;
	            #sx_ItemErrorMessageReq := TRUE;
	            #ii_ErrorNumber += 1;
	        ELSIF (#i_UDT_PDPStatus.Specific.CircuitBreakerTrippedF224 <> #s_UDT_PDPOldStatus.Specific.CircuitBreakerTrippedF224 AND NOT #sx_SendAllProcedure)
	            OR (#sx_SendAllProcedure AND #ii_ErrorNumber = 61)
	        THEN
	            #sdi_Code := "DB_MFC_ErrorCode".PDP.CircuitBreakerTrippedF224;
	            #si_State := BOOL_TO_INT(#i_UDT_PDPStatus.Specific.CircuitBreakerTrippedF224);
	            #s_UDT_PDPOldStatus.Specific.CircuitBreakerTrippedF224 := #i_UDT_PDPStatus.Specific.CircuitBreakerTrippedF224;
	            #sx_ItemErrorMessageReq := TRUE;
	            #ii_ErrorNumber += 1;
	        ELSIF (#i_UDT_PDPStatus.Specific.CircuitBreakerTrippedF225 <> #s_UDT_PDPOldStatus.Specific.CircuitBreakerTrippedF225 AND NOT #sx_SendAllProcedure)
	            OR (#sx_SendAllProcedure AND #ii_ErrorNumber = 62)
	        THEN
	            #sdi_Code := "DB_MFC_ErrorCode".PDP.CircuitBreakerTrippedF225;
	            #si_State := BOOL_TO_INT(#i_UDT_PDPStatus.Specific.CircuitBreakerTrippedF225);
	            #s_UDT_PDPOldStatus.Specific.CircuitBreakerTrippedF225 := #i_UDT_PDPStatus.Specific.CircuitBreakerTrippedF225;
	            #sx_ItemErrorMessageReq := TRUE;
	            #ii_ErrorNumber += 1;
	        ELSIF (#i_UDT_PDPStatus.Specific.CircuitBreakerTrippedF226 <> #s_UDT_PDPOldStatus.Specific.CircuitBreakerTrippedF226 AND NOT #sx_SendAllProcedure)
	            OR (#sx_SendAllProcedure AND #ii_ErrorNumber = 63)
	        THEN
	            #sdi_Code := "DB_MFC_ErrorCode".PDP.CircuitBreakerTrippedF226;
	            #si_State := BOOL_TO_INT(#i_UDT_PDPStatus.Specific.CircuitBreakerTrippedF226);
	            #s_UDT_PDPOldStatus.Specific.CircuitBreakerTrippedF226 := #i_UDT_PDPStatus.Specific.CircuitBreakerTrippedF226;
	            #sx_ItemErrorMessageReq := TRUE;
	            #ii_ErrorNumber += 1;
	        ELSIF (#i_UDT_PDPStatus.Specific.CircuitBreakerTrippedF227 <> #s_UDT_PDPOldStatus.Specific.CircuitBreakerTrippedF227 AND NOT #sx_SendAllProcedure)
	            OR (#sx_SendAllProcedure AND #ii_ErrorNumber = 64)
	        THEN
	            #sdi_Code := "DB_MFC_ErrorCode".PDP.CircuitBreakerTrippedF227;
	            #si_State := BOOL_TO_INT(#i_UDT_PDPStatus.Specific.CircuitBreakerTrippedF227);
	            #s_UDT_PDPOldStatus.Specific.CircuitBreakerTrippedF227 := #i_UDT_PDPStatus.Specific.CircuitBreakerTrippedF227;
	            #sx_ItemErrorMessageReq := TRUE;
	            #ii_ErrorNumber += 1;
	        ELSIF (#i_UDT_PDPStatus.Specific.CircuitBreakerTrippedF228 <> #s_UDT_PDPOldStatus.Specific.CircuitBreakerTrippedF228 AND NOT #sx_SendAllProcedure)
	            OR (#sx_SendAllProcedure AND #ii_ErrorNumber = 65)
	        THEN
	            #sdi_Code := "DB_MFC_ErrorCode".PDP.CircuitBreakerTrippedF228;
	            #si_State := BOOL_TO_INT(#i_UDT_PDPStatus.Specific.CircuitBreakerTrippedF228);
	            #s_UDT_PDPOldStatus.Specific.CircuitBreakerTrippedF228 := #i_UDT_PDPStatus.Specific.CircuitBreakerTrippedF228;
	            #sx_ItemErrorMessageReq := TRUE;
	            #ii_ErrorNumber += 1;
	        ELSIF (#i_UDT_PDPStatus.Specific.CircuitBreakerTrippedF229 <> #s_UDT_PDPOldStatus.Specific.CircuitBreakerTrippedF229 AND NOT #sx_SendAllProcedure)
	            OR (#sx_SendAllProcedure AND #ii_ErrorNumber = 66)
	        THEN
	            #sdi_Code := "DB_MFC_ErrorCode".PDP.CircuitBreakerTrippedF229;
	            #si_State := BOOL_TO_INT(#i_UDT_PDPStatus.Specific.CircuitBreakerTrippedF229);
	            #s_UDT_PDPOldStatus.Specific.CircuitBreakerTrippedF229 := #i_UDT_PDPStatus.Specific.CircuitBreakerTrippedF229;
	            #sx_ItemErrorMessageReq := TRUE;
	            #ii_ErrorNumber += 1;



	        ELSIF (#i_UDT_PDPStatus.Specific.CircuitBreakerTrippedF501 <> #s_UDT_PDPOldStatus.Specific.CircuitBreakerTrippedF501 AND NOT #sx_SendAllProcedure)
	            OR (#sx_SendAllProcedure AND #ii_ErrorNumber = 67)
	        THEN
	            #sdi_Code := "DB_MFC_ErrorCode".PDP.CircuitBreakerTrippedF501;
	            #si_State := BOOL_TO_INT(#i_UDT_PDPStatus.Specific.CircuitBreakerTrippedF501);
	            #s_UDT_PDPOldStatus.Specific.CircuitBreakerTrippedF501 := #i_UDT_PDPStatus.Specific.CircuitBreakerTrippedF501;
	            #sx_ItemErrorMessageReq := TRUE;
	            #ii_ErrorNumber += 1;
	        ELSIF (#i_UDT_PDPStatus.Specific.CircuitBreakerTrippedF502 <> #s_UDT_PDPOldStatus.Specific.CircuitBreakerTrippedF502 AND NOT #sx_SendAllProcedure)
	            OR (#sx_SendAllProcedure AND #ii_ErrorNumber = 68)
	        THEN
	            #sdi_Code := "DB_MFC_ErrorCode".PDP.CircuitBreakerTrippedF502;
	            #si_State := BOOL_TO_INT(#i_UDT_PDPStatus.Specific.CircuitBreakerTrippedF502);
	            #s_UDT_PDPOldStatus.Specific.CircuitBreakerTrippedF502 := #i_UDT_PDPStatus.Specific.CircuitBreakerTrippedF502;
	            #sx_ItemErrorMessageReq := TRUE;
	            #ii_ErrorNumber += 1;
	        ELSIF (#i_UDT_PDPStatus.Specific.CircuitBreakerTrippedF503 <> #s_UDT_PDPOldStatus.Specific.CircuitBreakerTrippedF503 AND NOT #sx_SendAllProcedure)
	            OR (#sx_SendAllProcedure AND #ii_ErrorNumber = 69)
	        THEN
	            #sdi_Code := "DB_MFC_ErrorCode".PDP.CircuitBreakerTrippedF503;
	            #si_State := BOOL_TO_INT(#i_UDT_PDPStatus.Specific.CircuitBreakerTrippedF503);
	            #s_UDT_PDPOldStatus.Specific.CircuitBreakerTrippedF503 := #i_UDT_PDPStatus.Specific.CircuitBreakerTrippedF503;
	            #sx_ItemErrorMessageReq := TRUE;
	            #ii_ErrorNumber += 1;
	        ELSIF (#i_UDT_PDPStatus.Specific.CircuitBreakerTrippedF504 <> #s_UDT_PDPOldStatus.Specific.CircuitBreakerTrippedF504 AND NOT #sx_SendAllProcedure)
	            OR (#sx_SendAllProcedure AND #ii_ErrorNumber = 70)
	        THEN
	            #sdi_Code := "DB_MFC_ErrorCode".PDP.CircuitBreakerTrippedF504;
	            #si_State := BOOL_TO_INT(#i_UDT_PDPStatus.Specific.CircuitBreakerTrippedF504);
	            #s_UDT_PDPOldStatus.Specific.CircuitBreakerTrippedF504 := #i_UDT_PDPStatus.Specific.CircuitBreakerTrippedF504;
	            #sx_ItemErrorMessageReq := TRUE;
	            #ii_ErrorNumber += 1;
	        ELSIF (#i_UDT_PDPStatus.Specific.CircuitBreakerTrippedF505 <> #s_UDT_PDPOldStatus.Specific.CircuitBreakerTrippedF505 AND NOT #sx_SendAllProcedure)
	            OR (#sx_SendAllProcedure AND #ii_ErrorNumber = 71)
	        THEN
	            #sdi_Code := "DB_MFC_ErrorCode".PDP.CircuitBreakerTrippedF505;
	            #si_State := BOOL_TO_INT(#i_UDT_PDPStatus.Specific.CircuitBreakerTrippedF505);
	            #s_UDT_PDPOldStatus.Specific.CircuitBreakerTrippedF505 := #i_UDT_PDPStatus.Specific.CircuitBreakerTrippedF505;
	            #sx_ItemErrorMessageReq := TRUE;
	            #ii_ErrorNumber += 1;
	        ELSIF (#i_UDT_PDPStatus.Specific.CircuitBreakerTrippedF506 <> #s_UDT_PDPOldStatus.Specific.CircuitBreakerTrippedF506 AND NOT #sx_SendAllProcedure)
	            OR (#sx_SendAllProcedure AND #ii_ErrorNumber = 72)
	        THEN
	            #sdi_Code := "DB_MFC_ErrorCode".PDP.CircuitBreakerTrippedF506;
	            #si_State := BOOL_TO_INT(#i_UDT_PDPStatus.Specific.CircuitBreakerTrippedF506);
	            #s_UDT_PDPOldStatus.Specific.CircuitBreakerTrippedF506 := #i_UDT_PDPStatus.Specific.CircuitBreakerTrippedF506;
	            #sx_ItemErrorMessageReq := TRUE;
	            #ii_ErrorNumber += 1;
	        ELSIF (#i_UDT_PDPStatus.Specific.CircuitBreakerTrippedF507 <> #s_UDT_PDPOldStatus.Specific.CircuitBreakerTrippedF507 AND NOT #sx_SendAllProcedure)
	            OR (#sx_SendAllProcedure AND #ii_ErrorNumber = 73)
	        THEN
	            #sdi_Code := "DB_MFC_ErrorCode".PDP.CircuitBreakerTrippedF507;
	            #si_State := BOOL_TO_INT(#i_UDT_PDPStatus.Specific.CircuitBreakerTrippedF507);
	            #s_UDT_PDPOldStatus.Specific.CircuitBreakerTrippedF507 := #i_UDT_PDPStatus.Specific.CircuitBreakerTrippedF507;
	            #sx_ItemErrorMessageReq := TRUE;
	            #ii_ErrorNumber += 1;
	        ELSIF (#i_UDT_PDPStatus.Specific.CircuitBreakerTrippedF508 <> #s_UDT_PDPOldStatus.Specific.CircuitBreakerTrippedF508 AND NOT #sx_SendAllProcedure)
	            OR (#sx_SendAllProcedure AND #ii_ErrorNumber = 74)
	        THEN
	            #sdi_Code := "DB_MFC_ErrorCode".PDP.CircuitBreakerTrippedF508;
	            #si_State := BOOL_TO_INT(#i_UDT_PDPStatus.Specific.CircuitBreakerTrippedF508);
	            #s_UDT_PDPOldStatus.Specific.CircuitBreakerTrippedF508 := #i_UDT_PDPStatus.Specific.CircuitBreakerTrippedF508;
	            #sx_ItemErrorMessageReq := TRUE;
	            #ii_ErrorNumber += 1;
	        ELSIF (#i_UDT_PDPStatus.Specific.CircuitBreakerTrippedF509 <> #s_UDT_PDPOldStatus.Specific.CircuitBreakerTrippedF509 AND NOT #sx_SendAllProcedure)
	            OR (#sx_SendAllProcedure AND #ii_ErrorNumber = 75)
	        THEN
	            #sdi_Code := "DB_MFC_ErrorCode".PDP.CircuitBreakerTrippedF509;
	            #si_State := BOOL_TO_INT(#i_UDT_PDPStatus.Specific.CircuitBreakerTrippedF509);
	            #s_UDT_PDPOldStatus.Specific.CircuitBreakerTrippedF509 := #i_UDT_PDPStatus.Specific.CircuitBreakerTrippedF509;
	            #sx_ItemErrorMessageReq := TRUE;
	            #ii_ErrorNumber += 1;
	        ELSIF (#i_UDT_PDPStatus.Specific.CircuitBreakerTrippedF510 <> #s_UDT_PDPOldStatus.Specific.CircuitBreakerTrippedF510 AND NOT #sx_SendAllProcedure)
	            OR (#sx_SendAllProcedure AND #ii_ErrorNumber = 76)
	        THEN
	            #sdi_Code := "DB_MFC_ErrorCode".PDP.CircuitBreakerTrippedF510;
	            #si_State := BOOL_TO_INT(#i_UDT_PDPStatus.Specific.CircuitBreakerTrippedF510);
	            #s_UDT_PDPOldStatus.Specific.CircuitBreakerTrippedF510 := #i_UDT_PDPStatus.Specific.CircuitBreakerTrippedF510;
	            #sx_ItemErrorMessageReq := TRUE;
	            #ii_ErrorNumber += 1;
	        ELSIF (#i_UDT_PDPStatus.Specific.CircuitBreakerTrippedF511 <> #s_UDT_PDPOldStatus.Specific.CircuitBreakerTrippedF511 AND NOT #sx_SendAllProcedure)
	            OR (#sx_SendAllProcedure AND #ii_ErrorNumber = 77)
	        THEN
	            #sdi_Code := "DB_MFC_ErrorCode".PDP.CircuitBreakerTrippedF511;
	            #si_State := BOOL_TO_INT(#i_UDT_PDPStatus.Specific.CircuitBreakerTrippedF511);
	            #s_UDT_PDPOldStatus.Specific.CircuitBreakerTrippedF511 := #i_UDT_PDPStatus.Specific.CircuitBreakerTrippedF511;
	            #sx_ItemErrorMessageReq := TRUE;
	            #ii_ErrorNumber += 1;
	        ELSIF (#i_UDT_PDPStatus.Specific.CircuitBreakerTrippedF512 <> #s_UDT_PDPOldStatus.Specific.CircuitBreakerTrippedF512 AND NOT #sx_SendAllProcedure)
	            OR (#sx_SendAllProcedure AND #ii_ErrorNumber = 78)
	        THEN
	            #sdi_Code := "DB_MFC_ErrorCode".PDP.CircuitBreakerTrippedF512;
	            #si_State := BOOL_TO_INT(#i_UDT_PDPStatus.Specific.CircuitBreakerTrippedF512);
	            #s_UDT_PDPOldStatus.Specific.CircuitBreakerTrippedF512 := #i_UDT_PDPStatus.Specific.CircuitBreakerTrippedF512;
	            #sx_ItemErrorMessageReq := TRUE;
	            #sx_SendAllProcedure := FALSE;
	            #ii_ErrorNumber += 1;
	        END_IF;
	    END_IF;
	END_REGION

	REGION 4 - Write message components to the item error structure

	    #s_UDT_ItemError.ItemNumber := #i_UDT_EquipmentNumber;
	    #s_UDT_ItemError.Error := #sdi_Code;
	    #s_UDT_ItemError.State := #si_State;
	    #s_UDT_ItemError.Masked := 1;

	END_REGION

	REGION 5 - Write message components to the item status structure

	    #s_UDT_ItemStatus.Group := #i_UDT_EquipmentNumber.Group;
	    #s_UDT_ItemStatus.Node := #i_UDT_EquipmentNumber.Node;
	    #s_UDT_ItemStatus.Status := #si_ItemStatus;

	END_REGION

	REGION 6 - Prepare messages to the MFC

	    // If item error message required signal is set, prepare the item error message.
	    IF (#sx_ItemErrorMessageReq)
	    THEN
	        #s_FB_ItemError(i_UDT_ItemErrorBody := #s_UDT_ItemError,
	                        ii_MessageGroup := 1,
	                        ix_FlagRetry := FALSE,
	                        idi_TimeSpan := 0,
	                        qx_Error => #sx_ItemErrorBlockError,
	                        qx_Warning => #sx_ItemErrorBlockWarning,
	                        iq_UDT_FifoHeader := #iq_UDT_FifoHeader,
	                        iqs_FifoData := #iqs_FifoData,
	                        iqdi_MessageSequenceNumber := #iqdi_MessageSequenceNumber);
	    END_IF;

	    // If item status message required signal is set, prepare the item error message.
	    IF (#sx_ItemStatusMessageReq)
	    THEN
	        #s_FB_ItemStatus(i_UDT_ItemStatusBody := #s_UDT_ItemStatus,
	                         ii_MessageGroup := 1,
	                         ix_FlagRetry := FALSE,
	                         idi_TimeSpan := 0,
	                         qx_Error => #sx_ItemStatusBlockError,
	                         qx_Warning => #sx_ItemStatusBlockWarning,
	                         iq_UDT_FifoHeader := #iq_UDT_FifoHeader,
	                         iqs_FifoData := #iqs_FifoData,
	                         iqdi_MessageSequenceNumber := #iqdi_MessageSequenceNumber);
	    END_IF;

	END_REGION

	REGION 7 - Write outputs

	    // Prepare collective output error.
	    #qx_Error :=
	    #sx_ItemErrorBlockError
	    OR #sx_ItemStatusBlockError
	    OR #sx_FIFOError;

	    // Prepare collective output warning.
	    #qx_Warning :=
	    #sx_ItemErrorBlockWarning
	    OR #sx_ItemStatusBlockWarning
	    OR #sx_FIFOWarning;

	END_REGION









END_FUNCTION_BLOCK

FUNCTION_BLOCK "FB_MFC_Visu_ABSwitch_Status"
{ S7_Optimized_Access := 'TRUE' }
VERSION : 0.1
// ATTRIBUTES
// AUTO_NUMBER = True
// BLOCK_NUMBER = 134
// END_ATTRIBUTES
   VAR_INPUT
      i_UDT_ABSwitchStatus { ExternalAccessible := 'False'; ExternalVisible := 'False'; ExternalWritable := 'False'} : "UDT_ABSwitchStatus";   // ColumnLift status structure
      i_UDT_EquipmentNumber { ExternalAccessible := 'False'; ExternalVisible := 'False'; ExternalWritable := 'False'} : "UDT_EquipmentNumber";   // Item number
      ix_SendAllErrorsState { ExternalAccessible := 'False'; ExternalVisible := 'False'; ExternalWritable := 'False'} : Bool;   // True - update all the messages
      ix_MFCConnected { ExternalAccessible := 'False'; ExternalVisible := 'False'; ExternalWritable := 'False'} : Bool;   // True - A connection to the MFC has been established
      ix_CollectiveReset { ExternalAccessible := 'False'; ExternalVisible := 'False'; ExternalWritable := 'False'} : Bool;   // True - Collective reset command of all system controls
   END_VAR

   VAR_OUTPUT
      qx_Error { ExternalAccessible := 'False'; ExternalVisible := 'False'; ExternalWritable := 'False'} : Bool;   // Block error
      qx_Warning { ExternalAccessible := 'False'; ExternalVisible := 'False'; ExternalWritable := 'False'} : Bool;   // Block warning
   END_VAR

   VAR_IN_OUT
      iq_UDT_FifoHeader : "UDT_FifoHeader";   // FIFO header
      iqs_FifoData : Array[*] of "UDT_MessageV2";   // FIFO data buffer
      iqdi_MessageSequenceNumber { ExternalAccessible := 'False'; ExternalVisible := 'False'; ExternalWritable := 'False'} : DInt;   // Message number
   END_VAR

   VAR
      s_FB_ItemError { ExternalAccessible := 'False'; ExternalVisible := 'False'; ExternalWritable := 'False'; S7_SetPoint := 'False'} : "FB_ItemError";   // Item error block's instance
      s_FB_ItemStatus { ExternalAccessible := 'False'; ExternalVisible := 'False'; ExternalWritable := 'False'; S7_SetPoint := 'False'} : "FB_ItemStatus";   // Item status block's instance
      ss_FIFOStatus { ExternalAccessible := 'False'; ExternalVisible := 'False'; ExternalWritable := 'False'; S7_SetPoint := 'False'} : "UDT_FifoStatus";   // Status structure
      s_UDT_Message { ExternalAccessible := 'False'; ExternalVisible := 'False'; ExternalWritable := 'False'; S7_SetPoint := 'False'} : "UDT_MessageV2";   // Message
      s_UDT_ABSwitch_StatusOld { ExternalAccessible := 'False'; ExternalVisible := 'False'; ExternalWritable := 'False'; S7_SetPoint := 'False'} : "UDT_ABSwitchStatus";   // ColumnLift status structure
      s_UDT_ItemError { ExternalAccessible := 'False'; ExternalVisible := 'False'; ExternalWritable := 'False'; S7_SetPoint := 'False'} : "UDT_ItemError";   // Item error message body structure
      s_UDT_ItemStatus { ExternalAccessible := 'False'; ExternalVisible := 'False'; ExternalWritable := 'False'; S7_SetPoint := 'False'} : "UDT_ItemStatus";   // Item status message body structure
      s_R_TRIG_Connection {InstructionName := 'R_TRIG'; LibVersion := '1.0'; ExternalAccessible := 'False'; ExternalVisible := 'False'; ExternalWritable := 'False'; S7_SetPoint := 'False'} : R_TRIG;   // Rising edge trigger connection reastablished
      s_F_TRIG_SendAllErrors {InstructionName := 'F_TRIG'; LibVersion := '1.0'; ExternalAccessible := 'False'; ExternalVisible := 'False'; ExternalWritable := 'False'; S7_SetPoint := 'False'} : F_TRIG;   // Falling edge trigger from signal send all errors
      sdi_Code { ExternalAccessible := 'False'; ExternalVisible := 'False'; ExternalWritable := 'False'} : DInt;   // Error code
      si_ItemStatus { ExternalAccessible := 'False'; ExternalVisible := 'False'; ExternalWritable := 'False'} : Int;   // Item status
      ii_ErrorNumber { ExternalAccessible := 'False'; ExternalVisible := 'False'; ExternalWritable := 'False'} : Int;   // Counter Error Number
      si_State { ExternalAccessible := 'False'; ExternalVisible := 'False'; ExternalWritable := 'False'} : Int;   // Error state
      sx_ItemErrorMessageReq { ExternalAccessible := 'False'; ExternalVisible := 'False'; ExternalWritable := 'False'} : Bool;   // Item error message required
      sx_ItemStatusMessageReq { ExternalAccessible := 'False'; ExternalVisible := 'False'; ExternalWritable := 'False'} : Bool;   // Item status message required
      sx_SendAllProcedure { ExternalAccessible := 'False'; ExternalVisible := 'False'; ExternalWritable := 'False'} : Bool;   // Send all procedure
      sx_FIFOError { ExternalAccessible := 'False'; ExternalVisible := 'False'; ExternalWritable := 'False'} : Bool;   // FIFO error
      sx_FIFOWarning { ExternalAccessible := 'False'; ExternalVisible := 'False'; ExternalWritable := 'False'} : Bool;   // FIFO warning
      sx_ItemErrorBlockError { ExternalAccessible := 'False'; ExternalVisible := 'False'; ExternalWritable := 'False'} : Bool;   // Item error block error
      sx_ItemErrorBlockWarning { ExternalAccessible := 'False'; ExternalVisible := 'False'; ExternalWritable := 'False'} : Bool;   // Item error block warning
      sx_ItemStatusBlockError { ExternalAccessible := 'False'; ExternalVisible := 'False'; ExternalWritable := 'False'} : Bool;   // Item status block error
      sx_ItemStatusBlockWarning { ExternalAccessible := 'False'; ExternalVisible := 'False'; ExternalWritable := 'False'} : Bool;   // Item status block warning
   END_VAR


BEGIN
	(*
	----------------------------------------------------------------------------------------
	|                                                                                      |
	|  Copyright  2023             FORTNA Europe BV                                        |
	|  All Rights Reserved         Netherlands                                             |
	|                                                                                      |
	----------------------------------------------------------------------------------------
	Version history:
	Date        | Version   | Author       | Remark
	----------------------------------------------------------------------------------------
	24/04/2023  | 1.0       | M. Diebel   | Release TIA 17 | DHL Munich 2023
	13/03/2023  | 1.1       | S. Nieswiec  | Updated for new Baseline
	*)


	REGION 1 - Initialize message required signals

	    #sx_ItemErrorMessageReq := FALSE;
	    #sx_ItemStatusMessageReq := FALSE;

	    // On connection reestablish send last remembered status and error state ( status only when it's diffrent then 0 )
	    #s_R_TRIG_Connection(CLK := #ix_MFCConnected);

	    IF #s_R_TRIG_Connection.Q AND #si_ItemStatus <> 0
	    THEN
	        #sx_ItemStatusMessageReq := TRUE;
	    END_IF;

	    IF #s_R_TRIG_Connection.Q
	    THEN
	        #sx_ItemErrorMessageReq := TRUE;
	    END_IF;

	    // Prepare trigger on the collective reset signal.
	    #s_F_TRIG_SendAllErrors(CLK := #ix_SendAllErrorsState);

	    // When collective reset will go down, start send every equipment errors.
	    IF #s_F_TRIG_SendAllErrors.Q AND NOT #sx_SendAllProcedure
	    THEN
	        #ii_ErrorNumber := 0;
	        #sx_SendAllProcedure := TRUE;
	    END_IF;

	END_REGION

	REGION 2 - FIFO header status update

	    // Mode 'S' - FIFO register status update.
	    "FC_Fifo"(ic_Mode := 'S',
	              qUDT_Status => #ss_FIFOStatus,
	              qx_Error => #sx_FIFOError,
	              qx_Warning => #sx_FIFOWarning,
	              iqv_Data := #s_UDT_Message,
	              iqUDT_FifoHeader := #iq_UDT_FifoHeader,
	              iqv_DataBuffer := #iqs_FifoData);

	END_REGION

	REGION 3 - Prepare message data

	    // When there is no reset errors command, update status and errors.
	    IF NOT #ix_CollectiveReset
	        AND NOT #ss_FIFOStatus.FifoPreFull
	    THEN
	        // Status
	        IF (#i_UDT_ABSwitchStatus.Status <> #s_UDT_ABSwitch_StatusOld.Status OR (#sx_SendAllProcedure AND #ii_ErrorNumber = 0))
	        THEN
	            #sx_ItemStatusMessageReq := TRUE;
	            #si_ItemStatus := #i_UDT_ABSwitchStatus.Status;
	            #s_UDT_ABSwitch_StatusOld.Status := #i_UDT_ABSwitchStatus.Status;
	        END_IF;


	        // Check which specific status changed, prepare code, change state and write new status into the old one.
	        IF (#i_UDT_ABSwitchStatus.Specific.ReferenceError <> #s_UDT_ABSwitch_StatusOld.Specific.ReferenceError AND NOT #sx_SendAllProcedure)
	            OR (#sx_SendAllProcedure AND #ii_ErrorNumber = 0)
	        THEN
	            #sdi_Code := "DB_MFC_ErrorCode".ABSwitch.ReferenceError;
	            #si_State := BOOL_TO_INT(#i_UDT_ABSwitchStatus.Specific.ReferenceError);
	            #s_UDT_ABSwitch_StatusOld.Specific.ReferenceError := #i_UDT_ABSwitchStatus.Specific.ReferenceError;
	            #sx_ItemErrorMessageReq := TRUE;
	            #ii_ErrorNumber += 1;
	        ELSIF (#i_UDT_ABSwitchStatus.Specific.SwitchingTimerError <> #s_UDT_ABSwitch_StatusOld.Specific.SwitchingTimerError AND NOT #sx_SendAllProcedure)
	            OR (#sx_SendAllProcedure AND #ii_ErrorNumber = 1)
	        THEN
	            #sdi_Code := "DB_MFC_ErrorCode".ABSwitch.SwitchingTimerError;
	            #si_State := BOOL_TO_INT(#i_UDT_ABSwitchStatus.Specific.SwitchingTimerError);
	            #s_UDT_ABSwitch_StatusOld.Specific.SwitchingTimerError := #i_UDT_ABSwitchStatus.Specific.SwitchingTimerError;
	            #sx_ItemErrorMessageReq := TRUE;
	            #ii_ErrorNumber += 1;
	        ELSIF (#i_UDT_ABSwitchStatus.Specific.LimitSensorUpperPosition <> #s_UDT_ABSwitch_StatusOld.Specific.LimitSensorUpperPosition AND NOT #sx_SendAllProcedure)
	            OR (#sx_SendAllProcedure AND #ii_ErrorNumber = 2)
	        THEN
	            #sdi_Code := "DB_MFC_ErrorCode".ABSwitch.LimitSensorUpperPosition;
	            #si_State := BOOL_TO_INT(#i_UDT_ABSwitchStatus.Specific.LimitSensorUpperPosition);
	            #s_UDT_ABSwitch_StatusOld.Specific.LimitSensorUpperPosition := #i_UDT_ABSwitchStatus.Specific.LimitSensorUpperPosition;
	            #sx_ItemErrorMessageReq := TRUE;
	            #ii_ErrorNumber += 1;
	        ELSIF (#i_UDT_ABSwitchStatus.Specific.LimitSensorLowerPosition <> #s_UDT_ABSwitch_StatusOld.Specific.LimitSensorLowerPosition AND NOT #sx_SendAllProcedure)
	            OR (#sx_SendAllProcedure AND #ii_ErrorNumber = 3)
	        THEN
	            #sdi_Code := "DB_MFC_ErrorCode".ABSwitch.LimitSensorLowerPosition;
	            #si_State := BOOL_TO_INT(#i_UDT_ABSwitchStatus.Specific.LimitSensorLowerPosition);
	            #s_UDT_ABSwitch_StatusOld.Specific.LimitSensorLowerPosition := #i_UDT_ABSwitchStatus.Specific.LimitSensorLowerPosition;
	            #sx_ItemErrorMessageReq := TRUE;
	            #ii_ErrorNumber += 1;
	        ELSIF (#i_UDT_ABSwitchStatus.Specific.UpperSwitchAreaError <> #s_UDT_ABSwitch_StatusOld.Specific.UpperSwitchAreaError AND NOT #sx_SendAllProcedure)
	            OR (#sx_SendAllProcedure AND #ii_ErrorNumber = 4)
	        THEN
	            #sdi_Code := "DB_MFC_ErrorCode".ABSwitch.UpperSwitchArea_Err;
	            #si_State := BOOL_TO_INT(#i_UDT_ABSwitchStatus.Specific.UpperSwitchAreaError);
	            #s_UDT_ABSwitch_StatusOld.Specific.UpperSwitchAreaError := #i_UDT_ABSwitchStatus.Specific.UpperSwitchAreaError;
	            #sx_ItemErrorMessageReq := TRUE;
	            #ii_ErrorNumber += 1;
	        ELSIF (#i_UDT_ABSwitchStatus.Specific.LowerSwitchAreaError <> #s_UDT_ABSwitch_StatusOld.Specific.LowerSwitchAreaError AND NOT #sx_SendAllProcedure)
	            OR (#sx_SendAllProcedure AND #ii_ErrorNumber = 5)
	        THEN
	            #sdi_Code := "DB_MFC_ErrorCode".ABSwitch.LowerSwitchArea_Err;
	            #si_State := BOOL_TO_INT(#i_UDT_ABSwitchStatus.Specific.LowerSwitchAreaError);
	            #s_UDT_ABSwitch_StatusOld.Specific.LowerSwitchAreaError := #i_UDT_ABSwitchStatus.Specific.LowerSwitchAreaError;
	            #sx_ItemErrorMessageReq := TRUE;
	            #ii_ErrorNumber += 1;
	        ELSIF (#i_UDT_ABSwitchStatus.Specific.UpperPosition <> #s_UDT_ABSwitch_StatusOld.Specific.UpperPosition AND NOT #sx_SendAllProcedure)
	            OR (#sx_SendAllProcedure AND #ii_ErrorNumber = 6)
	        THEN
	            #sdi_Code := "DB_MFC_ErrorCode".ABSwitch.UpperPosition;
	            #si_State := BOOL_TO_INT(#i_UDT_ABSwitchStatus.Specific.UpperPosition);
	            #s_UDT_ABSwitch_StatusOld.Specific.UpperPosition := #i_UDT_ABSwitchStatus.Specific.UpperPosition;
	            #sx_ItemErrorMessageReq := TRUE;
	            #ii_ErrorNumber += 1;
	        ELSIF (#i_UDT_ABSwitchStatus.Specific.LowerPosition <> #s_UDT_ABSwitch_StatusOld.Specific.LowerPosition AND NOT #sx_SendAllProcedure)
	            OR (#sx_SendAllProcedure AND #ii_ErrorNumber = 7)
	        THEN
	            #sdi_Code := "DB_MFC_ErrorCode".ABSwitch.LowerPosition;
	            #si_State := BOOL_TO_INT(#i_UDT_ABSwitchStatus.Specific.LowerPosition);
	            #s_UDT_ABSwitch_StatusOld.Specific.LowerPosition := #i_UDT_ABSwitchStatus.Specific.LowerPosition;
	            #sx_ItemErrorMessageReq := TRUE;
	            #sx_SendAllProcedure := FALSE;
	            #ii_ErrorNumber += 1;
	        END_IF;
	    END_IF;
	END_REGION

	REGION 4 - Write message components to the item error structure

	    #s_UDT_ItemError.ItemNumber := #i_UDT_EquipmentNumber;
	    #s_UDT_ItemError.Error := #sdi_Code;
	    #s_UDT_ItemError.State := #si_State;
	    #s_UDT_ItemError.Masked := 1;

	END_REGION

	REGION 5 - Write message components to the item status structure

	    #s_UDT_ItemStatus.Group := #i_UDT_EquipmentNumber.Group;
	    #s_UDT_ItemStatus.Node := #i_UDT_EquipmentNumber.Node;
	    #s_UDT_ItemStatus.Status := #si_ItemStatus;

	END_REGION

	REGION 6 - Prepare messages to the MFC

	    // If item error message required signal is set, prepare the item error message.
	    IF (#sx_ItemErrorMessageReq)
	    THEN
	        #s_FB_ItemError(i_UDT_ItemErrorBody := #s_UDT_ItemError,
	                        ii_MessageGroup := 1,
	                        ix_FlagRetry := FALSE,
	                        idi_TimeSpan := 0,
	                        qx_Error => #sx_ItemErrorBlockError,
	                        qx_Warning => #sx_ItemErrorBlockWarning,
	                        iq_UDT_FifoHeader := #iq_UDT_FifoHeader,
	                        iqs_FifoData := #iqs_FifoData,
	                        iqdi_MessageSequenceNumber := #iqdi_MessageSequenceNumber);
	    END_IF;

	    // If item status message required signal is set, prepare the item error message.
	    IF (#sx_ItemStatusMessageReq)
	    THEN
	        #s_FB_ItemStatus(i_UDT_ItemStatusBody := #s_UDT_ItemStatus,
	                         ii_MessageGroup := 1,
	                         ix_FlagRetry := FALSE,
	                         idi_TimeSpan := 0,
	                         qx_Error => #sx_ItemStatusBlockError,
	                         qx_Warning => #sx_ItemStatusBlockWarning,
	                         iq_UDT_FifoHeader := #iq_UDT_FifoHeader,
	                         iqs_FifoData := #iqs_FifoData,
	                         iqdi_MessageSequenceNumber := #iqdi_MessageSequenceNumber);
	    END_IF;

	END_REGION

	REGION 7 - Write outputs

	    // Prepare collective output error.
	    #qx_Error :=
	    #sx_ItemErrorBlockError
	    OR #sx_ItemStatusBlockError
	    OR #sx_FIFOError;

	    // Prepare collective output warning.
	    #qx_Warning :=
	    #sx_ItemErrorBlockWarning
	    OR #sx_ItemStatusBlockWarning
	    OR #sx_FIFOWarning;

	END_REGION
END_FUNCTION_BLOCK

FUNCTION_BLOCK "FB_MFC_Visu_MCP_Status"
{ S7_Optimized_Access := 'TRUE' }
VERSION : 0.1
// ATTRIBUTES
// AUTO_NUMBER = True
// BLOCK_NUMBER = 151
// END_ATTRIBUTES
   VAR_INPUT
      i_UDT_MCPStatus { ExternalAccessible := 'False'; ExternalVisible := 'False'; ExternalWritable := 'False'} : "UDT_MCPStatus";   // MCP status structure
      i_UDT_EquipmentNumber { ExternalAccessible := 'False'; ExternalVisible := 'False'; ExternalWritable := 'False'} : "UDT_EquipmentNumber";   // Item number
      ix_SendAllErrorsState { ExternalAccessible := 'False'; ExternalVisible := 'False'; ExternalWritable := 'False'} : Bool;   // True - update all the messages
      ix_MFCConnected { ExternalAccessible := 'False'; ExternalVisible := 'False'; ExternalWritable := 'False'} : Bool;   // True - A connection to the MFC has been established
      ix_CollectiveReset { ExternalAccessible := 'False'; ExternalVisible := 'False'; ExternalWritable := 'False'} : Bool;   // True - Collective reset command of all system controls
   END_VAR

   VAR_OUTPUT
      qx_Error { ExternalAccessible := 'False'; ExternalVisible := 'False'; ExternalWritable := 'False'} : Bool;   // Block error
      qx_Warning { ExternalAccessible := 'False'; ExternalVisible := 'False'; ExternalWritable := 'False'} : Bool;   // Block warning
   END_VAR

   VAR_IN_OUT
      iq_UDT_FifoHeader : "UDT_FifoHeader";   // FIFO header
      iqs_FifoData : Array[*] of "UDT_MessageV2";   // FIFO data buffer
      iqdi_MessageSequenceNumber { ExternalAccessible := 'False'; ExternalVisible := 'False'; ExternalWritable := 'False'} : DInt;   // Message number
   END_VAR

   VAR
      s_FB_ItemError { ExternalAccessible := 'False'; ExternalVisible := 'False'; ExternalWritable := 'False'; S7_SetPoint := 'False'} : "FB_ItemError";   // Item error block's instance
      s_FB_ItemStatus { ExternalAccessible := 'False'; ExternalVisible := 'False'; ExternalWritable := 'False'; S7_SetPoint := 'False'} : "FB_ItemStatus";   // Item status block's instance
      ss_FIFOStatus { ExternalAccessible := 'False'; ExternalVisible := 'False'; ExternalWritable := 'False'; S7_SetPoint := 'False'} : "UDT_FifoStatus";   // Status structure
      s_UDT_Message { ExternalAccessible := 'False'; ExternalVisible := 'False'; ExternalWritable := 'False'; S7_SetPoint := 'False'} : "UDT_MessageV2";   // Message
      s_UDT_MCPOld { ExternalAccessible := 'False'; ExternalVisible := 'False'; ExternalWritable := 'False'; S7_SetPoint := 'False'} : "UDT_MCPStatus";   // MCP old status structure
      s_UDT_ItemError { ExternalAccessible := 'False'; ExternalVisible := 'False'; ExternalWritable := 'False'; S7_SetPoint := 'False'} : "UDT_ItemError";   // Item error message body structure
      s_UDT_ItemStatus { ExternalAccessible := 'False'; ExternalVisible := 'False'; ExternalWritable := 'False'; S7_SetPoint := 'False'} : "UDT_ItemStatus";   // Item status message body structure
      s_R_TRIG_Connection {InstructionName := 'R_TRIG'; LibVersion := '1.0'; ExternalAccessible := 'False'; ExternalVisible := 'False'; ExternalWritable := 'False'; S7_SetPoint := 'False'} : R_TRIG;   // Rising edge trigger connection reastablished
      s_F_TRIG_SendAllErrors {InstructionName := 'F_TRIG'; LibVersion := '1.0'; ExternalAccessible := 'False'; ExternalVisible := 'False'; ExternalWritable := 'False'; S7_SetPoint := 'False'} : F_TRIG;   // Falling edge trigger from signal send all errors
      sdi_Code { ExternalAccessible := 'False'; ExternalVisible := 'False'; ExternalWritable := 'False'} : DInt;   // Error code
      ii_ErrorNumber { ExternalAccessible := 'False'; ExternalVisible := 'False'; ExternalWritable := 'False'} : Int;   // Counter Error Number
      si_ItemStatus { ExternalAccessible := 'False'; ExternalVisible := 'False'; ExternalWritable := 'False'} : Int;   // Item status
      si_State { ExternalAccessible := 'False'; ExternalVisible := 'False'; ExternalWritable := 'False'} : Int;   // Error state
      si_Rack { ExternalAccessible := 'False'; ExternalVisible := 'False'; ExternalWritable := 'False'} : Int;
      si_IOModule { ExternalAccessible := 'False'; ExternalVisible := 'False'; ExternalWritable := 'False'} : Int;
      sx_ItemErrorMessageReq { ExternalAccessible := 'False'; ExternalVisible := 'False'; ExternalWritable := 'False'} : Bool;   // Item error message required
      sx_ItemStatusMessageReq { ExternalAccessible := 'False'; ExternalVisible := 'False'; ExternalWritable := 'False'} : Bool;   // Item status message required
      sx_SendAllProcedure { ExternalAccessible := 'False'; ExternalVisible := 'False'; ExternalWritable := 'False'} : Bool;   // Send all procedure
      sx_FIFOError { ExternalAccessible := 'False'; ExternalVisible := 'False'; ExternalWritable := 'False'} : Bool;   // FIFO error
      sx_FIFOWarning { ExternalAccessible := 'False'; ExternalVisible := 'False'; ExternalWritable := 'False'} : Bool;   // FIFO warning
      sx_ItemErrorBlockError { ExternalAccessible := 'False'; ExternalVisible := 'False'; ExternalWritable := 'False'} : Bool;   // Item error block error
      sx_ItemErrorBlockWarning { ExternalAccessible := 'False'; ExternalVisible := 'False'; ExternalWritable := 'False'} : Bool;   // Item error block warning
      sx_ItemStatusBlockError { ExternalAccessible := 'False'; ExternalVisible := 'False'; ExternalWritable := 'False'} : Bool;   // Item status block error
      sx_ItemStatusBlockWarning { ExternalAccessible := 'False'; ExternalVisible := 'False'; ExternalWritable := 'False'} : Bool;   // Item status block warning
   END_VAR


BEGIN
	(*
	----------------------------------------------------------------------------------------
	|                                                                                      |
	|  Copyright  2023             FORTNA Europe BV                                        |
	|  All Rights Reserved         Netherlands                                             |
	|                                                                                      |
	----------------------------------------------------------------------------------------
	Version history:
	Date        | Version   | Author       | Remark
	----------------------------------------------------------------------------------------
	28/03/2023  | 1.0       | M. Diebel   | Release TIA 17 | DHL Munich 2023
	13/03/2023  | 1.1       | S. Nieswiec  | Updated for new Baseline
	*)


	REGION 1 - Initialize message required signals

	    #sx_ItemErrorMessageReq := FALSE;
	    #sx_ItemStatusMessageReq := FALSE;

	    // On connection reestablish send last remembered status and error state ( status only when it's diffrent then 0 )
	    #s_R_TRIG_Connection(CLK := #ix_MFCConnected);

	    IF #s_R_TRIG_Connection.Q AND #si_ItemStatus <> 0
	    THEN
	        #sx_ItemStatusMessageReq := TRUE;
	    END_IF;

	    IF #s_R_TRIG_Connection.Q
	    THEN
	        #sx_ItemErrorMessageReq := TRUE;
	    END_IF;

	    // Prepare trigger on the collective reset signal.
	    #s_F_TRIG_SendAllErrors(CLK := #ix_SendAllErrorsState);

	    // When collective reset will go down, start send every equipment errors.
	    IF #s_F_TRIG_SendAllErrors.Q AND NOT #sx_SendAllProcedure
	    THEN
	        #ii_ErrorNumber := 0;
	        #sx_SendAllProcedure := TRUE;
	    END_IF;

	END_REGION

	REGION 2 - FIFO header status update

	    // Mode 'S' - FIFO register status update.
	    "FC_Fifo"(ic_Mode := 'S',
	              qUDT_Status => #ss_FIFOStatus,
	              qx_Error => #sx_FIFOError,
	              qx_Warning => #sx_FIFOWarning,
	              iqv_Data := #s_UDT_Message,
	              iqUDT_FifoHeader := #iq_UDT_FifoHeader,
	              iqv_DataBuffer := #iqs_FifoData);

	END_REGION

	REGION 3 - Prepare message data

	    // When there is no reset errors command, update status and errors.
	    IF NOT #ix_CollectiveReset
	        AND NOT #ss_FIFOStatus.FifoPreFull
	    THEN
	        // Status
	        IF (#i_UDT_MCPStatus.Status <> #s_UDT_MCPOld.Status OR (#sx_SendAllProcedure AND #ii_ErrorNumber = 0))
	        THEN
	            #sx_ItemStatusMessageReq := TRUE;
	            #si_ItemStatus := #i_UDT_MCPStatus.Status;
	            #s_UDT_MCPOld.Status := #i_UDT_MCPStatus.Status;
	        END_IF;


	        // Check which specific status changed, prepare code, change state and write new status into the old one.
	        IF (#i_UDT_MCPStatus.Specific.PN_PN_MSP_PNSlaveNotOnline <> #s_UDT_MCPOld.Specific.PN_PN_MSP_PNSlaveNotOnline AND NOT #sx_SendAllProcedure)
	            OR (#sx_SendAllProcedure AND #ii_ErrorNumber = 0)
	        THEN
	            #sdi_Code := "DB_MFC_ErrorCode".MCP.PN_PN_MSP_PNSlaveNotOnline;
	            #si_State := BOOL_TO_INT(#i_UDT_MCPStatus.Specific.PN_PN_MSP_PNSlaveNotOnline);
	            #s_UDT_MCPOld.Specific.PN_PN_MSP_PNSlaveNotOnline := #i_UDT_MCPStatus.Specific.PN_PN_MSP_PNSlaveNotOnline;
	            #sx_ItemErrorMessageReq := TRUE;
	            #ii_ErrorNumber += 1;
	        ELSIF (#i_UDT_MCPStatus.Specific.PN_PN_MSP_PNSlaveError <> #s_UDT_MCPOld.Specific.PN_PN_MSP_PNSlaveError AND NOT #sx_SendAllProcedure)
	            OR (#sx_SendAllProcedure AND #ii_ErrorNumber = 1)
	        THEN
	            #sdi_Code := "DB_MFC_ErrorCode".MCP.PN_PN_MSP_PNSlaveError;
	            #si_State := BOOL_TO_INT(#i_UDT_MCPStatus.Specific.PN_PN_MSP_PNSlaveError);
	            #s_UDT_MCPOld.Specific.PN_PN_MSP_PNSlaveError := #i_UDT_MCPStatus.Specific.PN_PN_MSP_PNSlaveError;
	            #sx_ItemErrorMessageReq := TRUE;
	            #ii_ErrorNumber += 1;
	        ELSIF (#i_UDT_MCPStatus.Specific.PN_PN_MSP_PNSlaveWarning <> #s_UDT_MCPOld.Specific.PN_PN_MSP_PNSlaveWarning AND NOT #sx_SendAllProcedure)
	            OR (#sx_SendAllProcedure AND #ii_ErrorNumber = 2)
	        THEN
	            #sdi_Code := "DB_MFC_ErrorCode".MCP.PN_PN_MSP_PNSlaveWarning;
	            #si_State := BOOL_TO_INT(#i_UDT_MCPStatus.Specific.PN_PN_MSP_PNSlaveWarning);
	            #s_UDT_MCPOld.Specific.PN_PN_MSP_PNSlaveWarning := #i_UDT_MCPStatus.Specific.PN_PN_MSP_PNSlaveWarning;
	            #sx_ItemErrorMessageReq := TRUE;
	            #ii_ErrorNumber += 1;
	        ELSIF (#i_UDT_MCPStatus.Specific.IOModule_PNSlaveNotOnline <> #s_UDT_MCPOld.Specific.IOModule_PNSlaveNotOnline AND NOT #sx_SendAllProcedure)
	            OR (#sx_SendAllProcedure AND #ii_ErrorNumber = 3)
	        THEN
	            #sdi_Code := "DB_MFC_ErrorCode".MCP.IOModule_PNSlaveNotOnline;
	            #si_State := BOOL_TO_INT(#i_UDT_MCPStatus.Specific.IOModule_PNSlaveNotOnline);
	            #s_UDT_MCPOld.Specific.IOModule_PNSlaveNotOnline := #i_UDT_MCPStatus.Specific.IOModule_PNSlaveNotOnline;
	            #sx_ItemErrorMessageReq := TRUE;
	            #ii_ErrorNumber += 1;
	        ELSIF (#i_UDT_MCPStatus.Specific.IOModule_PNSlaveError <> #s_UDT_MCPOld.Specific.IOModule_PNSlaveError AND NOT #sx_SendAllProcedure)
	            OR (#sx_SendAllProcedure AND #ii_ErrorNumber = 4)
	        THEN
	            #sdi_Code := "DB_MFC_ErrorCode".MCP.IOModule_PNSlaveError;
	            #si_State := BOOL_TO_INT(#i_UDT_MCPStatus.Specific.IOModule_PNSlaveError);
	            #s_UDT_MCPOld.Specific.IOModule_PNSlaveError := #i_UDT_MCPStatus.Specific.IOModule_PNSlaveError;
	            #sx_ItemErrorMessageReq := TRUE;
	            #ii_ErrorNumber += 1;
	        ELSIF (#i_UDT_MCPStatus.Specific.IOModule_PNSlaveWarning <> #s_UDT_MCPOld.Specific.IOModule_PNSlaveWarning AND NOT #sx_SendAllProcedure)
	            OR (#sx_SendAllProcedure AND #ii_ErrorNumber = 5)
	        THEN
	            #sdi_Code := "DB_MFC_ErrorCode".MCP.IOModule_PNSlaveWarning;
	            #si_State := BOOL_TO_INT(#i_UDT_MCPStatus.Specific.IOModule_PNSlaveWarning);
	            #s_UDT_MCPOld.Specific.IOModule_PNSlaveWarning := #i_UDT_MCPStatus.Specific.IOModule_PNSlaveWarning;
	            #sx_ItemErrorMessageReq := TRUE;
	            #ii_ErrorNumber += 1;
	        ELSIF (#i_UDT_MCPStatus.Specific.ScalanceSwitchPNSlaveNotOnline <> #s_UDT_MCPOld.Specific.ScalanceSwitchPNSlaveNotOnline AND NOT #sx_SendAllProcedure)
	            OR (#sx_SendAllProcedure AND #ii_ErrorNumber = 6)
	        THEN
	            #sdi_Code := "DB_MFC_ErrorCode".MCP.ScalanceSwitchPNSlaveNotOnline;
	            #si_State := BOOL_TO_INT(#i_UDT_MCPStatus.Specific.ScalanceSwitchPNSlaveNotOnline);
	            #s_UDT_MCPOld.Specific.ScalanceSwitchPNSlaveNotOnline := #i_UDT_MCPStatus.Specific.ScalanceSwitchPNSlaveNotOnline;
	            #sx_ItemErrorMessageReq := TRUE;
	            #ii_ErrorNumber += 1;
	        ELSIF (#i_UDT_MCPStatus.Specific.ScalanceSwitchPNSlaveError <> #s_UDT_MCPOld.Specific.ScalanceSwitchPNSlaveError AND NOT #sx_SendAllProcedure)
	            OR (#sx_SendAllProcedure AND #ii_ErrorNumber = 7)
	        THEN
	            #sdi_Code := "DB_MFC_ErrorCode".MCP.ScalanceSwitchPNSlaveError;
	            #si_State := BOOL_TO_INT(#i_UDT_MCPStatus.Specific.ScalanceSwitchPNSlaveError);
	            #s_UDT_MCPOld.Specific.ScalanceSwitchPNSlaveError := #i_UDT_MCPStatus.Specific.ScalanceSwitchPNSlaveError;
	            #sx_ItemErrorMessageReq := TRUE;
	            #ii_ErrorNumber += 1;
	        ELSIF (#i_UDT_MCPStatus.Specific.ScalanceSwitchPNSlaveWarning <> #s_UDT_MCPOld.Specific.ScalanceSwitchPNSlaveWarning AND NOT #sx_SendAllProcedure)
	            OR (#sx_SendAllProcedure AND #ii_ErrorNumber = 8)
	        THEN
	            #sdi_Code := "DB_MFC_ErrorCode".MCP.ScalanceSwitchPNSlaveWarning;
	            #si_State := BOOL_TO_INT(#i_UDT_MCPStatus.Specific.ScalanceSwitchPNSlaveWarning);
	            #s_UDT_MCPOld.Specific.ScalanceSwitchPNSlaveWarning := #i_UDT_MCPStatus.Specific.ScalanceSwitchPNSlaveWarning;
	            #sx_ItemErrorMessageReq := TRUE;
	            #ii_ErrorNumber += 1;
	        ELSIF (#i_UDT_MCPStatus.Specific."2ndScalanceSwitchPNSlaveNotOnline" <> #s_UDT_MCPOld.Specific."2ndScalanceSwitchPNSlaveNotOnline" AND NOT #sx_SendAllProcedure)
	            OR (#sx_SendAllProcedure AND #ii_ErrorNumber = 9)
	        THEN
	            #sdi_Code := "DB_MFC_ErrorCode".MCP."2ndScalanceSwitchPNSlaveNotOnline";
	            #si_State := BOOL_TO_INT(#i_UDT_MCPStatus.Specific."2ndScalanceSwitchPNSlaveNotOnline");
	            #s_UDT_MCPOld.Specific."2ndScalanceSwitchPNSlaveNotOnline" := #i_UDT_MCPStatus.Specific."2ndScalanceSwitchPNSlaveNotOnline";
	            #sx_ItemErrorMessageReq := TRUE;
	            #ii_ErrorNumber += 1;
	        ELSIF (#i_UDT_MCPStatus.Specific."2ndScalanceSwitchPNSlaveError" <> #s_UDT_MCPOld.Specific."2ndScalanceSwitchPNSlaveError" AND NOT #sx_SendAllProcedure)
	            OR (#sx_SendAllProcedure AND #ii_ErrorNumber = 10)
	        THEN
	            #sdi_Code := "DB_MFC_ErrorCode".MCP."2ndScalanceSwitchPNSlaveError";
	            #si_State := BOOL_TO_INT(#i_UDT_MCPStatus.Specific."2ndScalanceSwitchPNSlaveError");
	            #s_UDT_MCPOld.Specific."2ndScalanceSwitchPNSlaveError" := #i_UDT_MCPStatus.Specific."2ndScalanceSwitchPNSlaveError";
	            #sx_ItemErrorMessageReq := TRUE;
	            #ii_ErrorNumber += 1;
	        ELSIF (#i_UDT_MCPStatus.Specific."2ndScalanceSwitchPNSlaveWarning" <> #s_UDT_MCPOld.Specific."2ndScalanceSwitchPNSlaveWarning" AND NOT #sx_SendAllProcedure)
	            OR (#sx_SendAllProcedure AND #ii_ErrorNumber = 11)
	        THEN
	            #sdi_Code := "DB_MFC_ErrorCode".MCP."2ndScalanceSwitchPNSlaveWarning";
	            #si_State := BOOL_TO_INT(#i_UDT_MCPStatus.Specific."2ndScalanceSwitchPNSlaveWarning");
	            #s_UDT_MCPOld.Specific."2ndScalanceSwitchPNSlaveWarning" := #i_UDT_MCPStatus.Specific."2ndScalanceSwitchPNSlaveWarning";
	            #sx_ItemErrorMessageReq := TRUE;
	            #ii_ErrorNumber += 1;
	        ELSIF (#i_UDT_MCPStatus.Specific.Singulator_PNSlaveNotOnline <> #s_UDT_MCPOld.Specific.Singulator_PNSlaveNotOnline AND NOT #sx_SendAllProcedure)
	            OR (#sx_SendAllProcedure AND #ii_ErrorNumber = 12)
	        THEN
	            #sdi_Code := "DB_MFC_ErrorCode".MCP.Singulator_PNSlaveNotOnline;
	            #si_State := BOOL_TO_INT(#i_UDT_MCPStatus.Specific.Singulator_PNSlaveNotOnline);
	            #s_UDT_MCPOld.Specific.Singulator_PNSlaveNotOnline := #i_UDT_MCPStatus.Specific.Singulator_PNSlaveNotOnline;
	            #sx_ItemErrorMessageReq := TRUE;
	            #ii_ErrorNumber += 1;
	        ELSIF (#i_UDT_MCPStatus.Specific.Singulator_PNSlaveError <> #s_UDT_MCPOld.Specific.Singulator_PNSlaveError AND NOT #sx_SendAllProcedure)
	            OR (#sx_SendAllProcedure AND #ii_ErrorNumber = 13)
	        THEN
	            #sdi_Code := "DB_MFC_ErrorCode".MCP.Singulator_PNSlaveError;
	            #si_State := BOOL_TO_INT(#i_UDT_MCPStatus.Specific.Singulator_PNSlaveError);
	            #s_UDT_MCPOld.Specific.Singulator_PNSlaveError := #i_UDT_MCPStatus.Specific.Singulator_PNSlaveError;
	            #sx_ItemErrorMessageReq := TRUE;
	            #ii_ErrorNumber += 1;
	        ELSIF (#i_UDT_MCPStatus.Specific.Singulator_PNSlaveWarning <> #s_UDT_MCPOld.Specific.Singulator_PNSlaveWarning AND NOT #sx_SendAllProcedure)
	            OR (#sx_SendAllProcedure AND #ii_ErrorNumber = 14)
	        THEN
	            #sdi_Code := "DB_MFC_ErrorCode".MCP.Singulator_PNSlaveWarning;
	            #si_State := BOOL_TO_INT(#i_UDT_MCPStatus.Specific.Singulator_PNSlaveWarning);
	            #s_UDT_MCPOld.Specific.Singulator_PNSlaveWarning := #i_UDT_MCPStatus.Specific.Singulator_PNSlaveWarning;
	            #sx_ItemErrorMessageReq := TRUE;
	            #ii_ErrorNumber += 1;
	        ELSIF (#i_UDT_MCPStatus.Specific.IPC_PNSlaveNotOnline <> #s_UDT_MCPOld.Specific.IPC_PNSlaveNotOnline AND NOT #sx_SendAllProcedure)
	            OR (#sx_SendAllProcedure AND #ii_ErrorNumber = 15)
	        THEN
	            #sdi_Code := "DB_MFC_ErrorCode".MCP.IPS_PNSlaveNotOnline;
	            #si_State := BOOL_TO_INT(#i_UDT_MCPStatus.Specific.IPC_PNSlaveNotOnline);
	            #s_UDT_MCPOld.Specific.IPC_PNSlaveNotOnline := #i_UDT_MCPStatus.Specific.IPC_PNSlaveNotOnline;
	            #sx_ItemErrorMessageReq := TRUE;
	            #ii_ErrorNumber += 1;
	        ELSIF (#i_UDT_MCPStatus.Specific.IPC_PNSlaveError <> #s_UDT_MCPOld.Specific.IPC_PNSlaveError AND NOT #sx_SendAllProcedure)
	            OR (#sx_SendAllProcedure AND #ii_ErrorNumber = 16)
	        THEN
	            #sdi_Code := "DB_MFC_ErrorCode".MCP.IPS_PNSlaveError;
	            #si_State := BOOL_TO_INT(#i_UDT_MCPStatus.Specific.IPC_PNSlaveError);
	            #s_UDT_MCPOld.Specific.IPC_PNSlaveError := #i_UDT_MCPStatus.Specific.IPC_PNSlaveError;
	            #sx_ItemErrorMessageReq := TRUE;
	            #ii_ErrorNumber += 1;
	        ELSIF (#i_UDT_MCPStatus.Specific.IPC_PNSlaveWarning <> #s_UDT_MCPOld.Specific.IPC_PNSlaveWarning AND NOT #sx_SendAllProcedure)
	            OR (#sx_SendAllProcedure AND #ii_ErrorNumber = 17)
	        THEN
	            #sdi_Code := "DB_MFC_ErrorCode".MCP.IPS_PNSlaveWarning;
	            #si_State := BOOL_TO_INT(#i_UDT_MCPStatus.Specific.IPC_PNSlaveWarning);
	            #s_UDT_MCPOld.Specific.IPC_PNSlaveWarning := #i_UDT_MCPStatus.Specific.IPC_PNSlaveWarning;
	            #sx_ItemErrorMessageReq := TRUE;
	            #ii_ErrorNumber += 1;
	        ELSIF (#i_UDT_MCPStatus.Specific.UPSSwitchTripped <> #s_UDT_MCPOld.Specific.UPSSwitchTripped AND NOT #sx_SendAllProcedure)
	            OR (#sx_SendAllProcedure AND #ii_ErrorNumber = 18)
	        THEN
	            #sdi_Code := "DB_MFC_ErrorCode".MCP.UPSSwitchTripped;
	            #si_State := BOOL_TO_INT(#i_UDT_MCPStatus.Specific.UPSSwitchTripped);
	            #s_UDT_MCPOld.Specific.UPSSwitchTripped := #i_UDT_MCPStatus.Specific.UPSSwitchTripped;
	            #sx_ItemErrorMessageReq := TRUE;
	            #ii_ErrorNumber += 1;
	        ELSIF (#i_UDT_MCPStatus.Specific.FireAlarmActive <> #s_UDT_MCPOld.Specific.FireAlarmActive AND NOT #sx_SendAllProcedure)
	            OR (#sx_SendAllProcedure AND #ii_ErrorNumber = 19)
	        THEN
	            #sdi_Code := "DB_MFC_ErrorCode".MCP.FireAlarmActive;
	            #si_State := BOOL_TO_INT(#i_UDT_MCPStatus.Specific.FireAlarmActive);
	            #s_UDT_MCPOld.Specific.FireAlarmActive := #i_UDT_MCPStatus.Specific.FireAlarmActive;
	            #sx_ItemErrorMessageReq := TRUE;
	            #ii_ErrorNumber += 1;
	        ELSIF (#i_UDT_MCPStatus.Specific.PS_201T1_Tripped <> #s_UDT_MCPOld.Specific.PS_201T1_Tripped AND NOT #sx_SendAllProcedure)
	            OR (#sx_SendAllProcedure AND #ii_ErrorNumber = 20)
	        THEN
	            #sdi_Code := "DB_MFC_ErrorCode".MCP.PS_201T1_Tripped;
	            #si_State := BOOL_TO_INT(#i_UDT_MCPStatus.Specific.PS_201T1_Tripped);
	            #s_UDT_MCPOld.Specific.PS_201T1_Tripped := #i_UDT_MCPStatus.Specific.PS_201T1_Tripped;
	            #sx_ItemErrorMessageReq := TRUE;
	            #ii_ErrorNumber += 1;
	        ELSIF (#i_UDT_MCPStatus.Specific."230VAC_CB101F4Tripped" <> #s_UDT_MCPOld.Specific."230VAC_CB101F4Tripped" AND NOT #sx_SendAllProcedure)
	            OR (#sx_SendAllProcedure AND #ii_ErrorNumber = 21)
	        THEN
	            #sdi_Code := "DB_MFC_ErrorCode".MCP."230VAC_CB101F4Tripped";
	            #si_State := BOOL_TO_INT(#i_UDT_MCPStatus.Specific."230VAC_CB101F4Tripped");
	            #s_UDT_MCPOld.Specific."230VAC_CB101F4Tripped" := #i_UDT_MCPStatus.Specific."230VAC_CB101F4Tripped";
	            #sx_ItemErrorMessageReq := TRUE;
	            #ii_ErrorNumber += 1;
	        ELSIF (#i_UDT_MCPStatus.Specific."230VAC_CB102F1Tripped" <> #s_UDT_MCPOld.Specific."230VAC_CB102F1Tripped" AND NOT #sx_SendAllProcedure)
	            OR (#sx_SendAllProcedure AND #ii_ErrorNumber = 22)
	        THEN
	            #sdi_Code := "DB_MFC_ErrorCode".MCP."230VAC_CB102F1Tripped";
	            #si_State := BOOL_TO_INT(#i_UDT_MCPStatus.Specific."230VAC_CB102F1Tripped");
	            #s_UDT_MCPOld.Specific."230VAC_CB102F1Tripped" := #i_UDT_MCPStatus.Specific."230VAC_CB102F1Tripped";
	            #sx_ItemErrorMessageReq := TRUE;
	            #ii_ErrorNumber += 1;
	        ELSIF (#i_UDT_MCPStatus.Specific."24VDC_CB201F1Tripped" <> #s_UDT_MCPOld.Specific."24VDC_CB201F1Tripped" AND NOT #sx_SendAllProcedure)
	            OR (#sx_SendAllProcedure AND #ii_ErrorNumber = 23)
	        THEN
	            #sdi_Code := "DB_MFC_ErrorCode".MCP."24VDC_CB201F1Tripped";
	            #si_State := BOOL_TO_INT(#i_UDT_MCPStatus.Specific."24VDC_CB201F1Tripped");
	            #s_UDT_MCPOld.Specific."24VDC_CB201F1Tripped" := #i_UDT_MCPStatus.Specific."24VDC_CB201F1Tripped";
	            #sx_ItemErrorMessageReq := TRUE;
	            #ii_ErrorNumber += 1;
	        ELSIF (#i_UDT_MCPStatus.Specific."24VDC_CB205F5Tripped" <> #s_UDT_MCPOld.Specific."24VDC_CB205F5Tripped" AND NOT #sx_SendAllProcedure)
	            OR (#sx_SendAllProcedure AND #ii_ErrorNumber = 24)
	        THEN
	            #sdi_Code := "DB_MFC_ErrorCode".MCP."24VDC_CB205F5Tripped";
	            #si_State := BOOL_TO_INT(#i_UDT_MCPStatus.Specific."24VDC_CB205F5Tripped");
	            #s_UDT_MCPOld.Specific."24VDC_CB205F5Tripped" := #i_UDT_MCPStatus.Specific."24VDC_CB205F5Tripped";
	            #sx_ItemErrorMessageReq := TRUE;
	            #sx_SendAllProcedure := FALSE;
	        ELSIF (#i_UDT_MCPStatus.Specific.Spare_1 <> #s_UDT_MCPOld.Specific.Spare_1 AND NOT #sx_SendAllProcedure)
	            OR (#sx_SendAllProcedure AND #ii_ErrorNumber = 25)
	        THEN
	            #sdi_Code := "DB_MFC_ErrorCode".MCP.Spare_1;
	            #si_State := BOOL_TO_INT(#i_UDT_MCPStatus.Specific.Spare_1);
	            #s_UDT_MCPOld.Specific.Spare_1 := #i_UDT_MCPStatus.Specific.Spare_1;
	            #sx_ItemErrorMessageReq := TRUE;
	        ELSIF (#i_UDT_MCPStatus.Specific.Spare_2 <> #s_UDT_MCPOld.Specific.Spare_2 AND NOT #sx_SendAllProcedure)
	            OR (#sx_SendAllProcedure AND #ii_ErrorNumber = 26)
	        THEN
	            #sdi_Code := "DB_MFC_ErrorCode".MCP.Spare_2;
	            #si_State := BOOL_TO_INT(#i_UDT_MCPStatus.Specific.Spare_2);
	            #s_UDT_MCPOld.Specific.Spare_2 := #i_UDT_MCPStatus.Specific.Spare_2;
	            #sx_ItemErrorMessageReq := TRUE;
	        ELSIF (#i_UDT_MCPStatus.Specific.Spare_3 <> #s_UDT_MCPOld.Specific.Spare_3 AND NOT #sx_SendAllProcedure)
	            OR (#sx_SendAllProcedure AND #ii_ErrorNumber = 27)
	        THEN
	            #sdi_Code := "DB_MFC_ErrorCode".MCP.Spare_3;
	            #si_State := BOOL_TO_INT(#i_UDT_MCPStatus.Specific.Spare_3);
	            #s_UDT_MCPOld.Specific.Spare_3 := #i_UDT_MCPStatus.Specific.Spare_3;
	            #sx_ItemErrorMessageReq := TRUE;
	            #sx_SendAllProcedure := FALSE;
	        ELSIF (#i_UDT_MCPStatus.Specific.RackSlotError <> #s_UDT_MCPOld.Specific.RackSlotError)
	        THEN
	            FOR #si_Rack := 0 TO 31 DO
	                IF (#i_UDT_MCPStatus.Specific.RackSlotError[#si_Rack] <> #s_UDT_MCPOld.Specific.RackSlotError[#si_Rack])
	                THEN
	                    #sdi_Code := "DB_MFC_ErrorCode".MCP.RackSlotError[#si_Rack];
	                    #si_State := BOOL_TO_INT(#i_UDT_MCPStatus.Specific.RackSlotError[#si_Rack]);
	                    #s_UDT_MCPOld.Specific.RackSlotError[#si_Rack] := #i_UDT_MCPStatus.Specific.RackSlotError[#si_Rack];
	                    #sx_ItemErrorMessageReq := TRUE;
	                    EXIT;
	                END_IF;
	            END_FOR;

	        ELSE

	            FOR #si_IOModule := 0 TO 31 DO
	                IF (#i_UDT_MCPStatus.Specific.IOModuleSlotError[#si_IOModule] <> #s_UDT_MCPOld.Specific.IOModuleSlotError[#si_IOModule])
	                THEN
	                    #sdi_Code := "DB_MFC_ErrorCode".MCP.IOModuleSlotError[#si_IOModule];
	                    #si_State := BOOL_TO_INT(#i_UDT_MCPStatus.Specific.IOModuleSlotError[#si_IOModule]);
	                    #s_UDT_MCPOld.Specific.IOModuleSlotError[#si_IOModule] := #i_UDT_MCPStatus.Specific.IOModuleSlotError[#si_IOModule];
	                    #sx_ItemErrorMessageReq := TRUE;
	                    EXIT;
	                END_IF;
	            END_FOR;

	        END_IF;
	    END_IF;
	END_REGION

	REGION 4 - Write message components to the item error structure

	    #s_UDT_ItemError.ItemNumber := #i_UDT_EquipmentNumber;
	    #s_UDT_ItemError.Error := #sdi_Code;
	    #s_UDT_ItemError.State := #si_State;
	    #s_UDT_ItemError.Masked := 1;

	END_REGION

	REGION 5 - Write message components to the item status structure

	    #s_UDT_ItemStatus.Group := #i_UDT_EquipmentNumber.Group;
	    #s_UDT_ItemStatus.Node := #i_UDT_EquipmentNumber.Node;
	    #s_UDT_ItemStatus.Status := #si_ItemStatus;

	END_REGION

	REGION 6 - Prepare messages to the MFC

	    // If item error message required signal is set, prepare the item error message.
	    IF (#sx_ItemErrorMessageReq)
	    THEN
	        #s_FB_ItemError(i_UDT_ItemErrorBody := #s_UDT_ItemError,
	                        ii_MessageGroup := 1,
	                        ix_FlagRetry := FALSE,
	                        idi_TimeSpan := 0,
	                        qx_Error => #sx_ItemErrorBlockError,
	                        qx_Warning => #sx_ItemErrorBlockWarning,
	                        iq_UDT_FifoHeader := #iq_UDT_FifoHeader,
	                        iqs_FifoData := #iqs_FifoData,
	                        iqdi_MessageSequenceNumber := #iqdi_MessageSequenceNumber);
	    END_IF;

	    // If item status message required signal is set, prepare the item error message.
	    IF (#sx_ItemStatusMessageReq)
	    THEN
	        #s_FB_ItemStatus(i_UDT_ItemStatusBody := #s_UDT_ItemStatus,
	                         ii_MessageGroup := 1,
	                         ix_FlagRetry := FALSE,
	                         idi_TimeSpan := 0,
	                         qx_Error => #sx_ItemStatusBlockError,
	                         qx_Warning => #sx_ItemStatusBlockWarning,
	                         iq_UDT_FifoHeader := #iq_UDT_FifoHeader,
	                         iqs_FifoData := #iqs_FifoData,
	                         iqdi_MessageSequenceNumber := #iqdi_MessageSequenceNumber);
	    END_IF;

	END_REGION

	REGION 7 - Write outputs

	    // Prepare collective output error.
	    #qx_Error :=
	    #sx_ItemErrorBlockError
	    OR #sx_ItemStatusBlockError
	    OR #sx_FIFOError;

	    // Prepare collective output warning.
	    #qx_Warning :=
	    #sx_ItemErrorBlockWarning
	    OR #sx_ItemStatusBlockWarning
	    OR #sx_FIFOWarning;

	END_REGION
END_FUNCTION_BLOCK

FUNCTION_BLOCK "FB_MFC_Visu_PEC_Status"
{ S7_Optimized_Access := 'TRUE' }
VERSION : 0.1
// ATTRIBUTES
// AUTO_NUMBER = True
// BLOCK_NUMBER = 154
// END_ATTRIBUTES
   VAR_INPUT
      ix_SendAllErrorsState { ExternalAccessible := 'False'; ExternalVisible := 'False'; ExternalWritable := 'False'} : Bool;   // True - update all the messages
      ix_MFCConnected { ExternalAccessible := 'False'; ExternalVisible := 'False'; ExternalWritable := 'False'} : Bool;   // True - A connection to the MFC has been established
      ix_CollectiveReset { ExternalAccessible := 'False'; ExternalVisible := 'False'; ExternalWritable := 'False'} : Bool;   // True - Collective reset command of all system controls
      i_UDT_PECStatus { ExternalAccessible := 'False'; ExternalVisible := 'False'; ExternalWritable := 'False'} : "UDT_PECStatus";   // PEC status structrue
      i_UDT_EquipmentNumber { ExternalAccessible := 'False'; ExternalVisible := 'False'; ExternalWritable := 'False'} : "UDT_EquipmentNumber";   // Equipment Number
   END_VAR

   VAR_OUTPUT
      qx_Error { ExternalAccessible := 'False'; ExternalVisible := 'False'; ExternalWritable := 'False'} : Bool;   // Block error
      qx_Warning { ExternalAccessible := 'False'; ExternalVisible := 'False'; ExternalWritable := 'False'} : Bool;   // Block warning
   END_VAR

   VAR_IN_OUT
      iq_UDT_FifoHeader : "UDT_FifoHeader";   // FIFO header
      iqs_FifoData : Array[*] of "UDT_MessageV2";   // FIFO data buffer
      iqdi_MessageSequenceNumber { ExternalAccessible := 'False'; ExternalVisible := 'False'; ExternalWritable := 'False'} : DInt;   // Message number
   END_VAR

   VAR
      s_FB_ItemError { ExternalAccessible := 'False'; ExternalVisible := 'False'; ExternalWritable := 'False'; S7_SetPoint := 'False'} : "FB_ItemError";   // Item error block instance
      s_UDT_Message { ExternalAccessible := 'False'; ExternalVisible := 'False'; ExternalWritable := 'False'; S7_SetPoint := 'False'} : "UDT_BytesMessage";   // Message
      s_UDT_ItemError { ExternalAccessible := 'False'; ExternalVisible := 'False'; ExternalWritable := 'False'; S7_SetPoint := 'False'} : "UDT_ItemError";   // Item error message body structure
      s_UDT_PECOLD { ExternalAccessible := 'False'; ExternalVisible := 'False'; ExternalWritable := 'False'; S7_SetPoint := 'False'} : "UDT_PECStatus";   // PEC old status structure
      s_UDT_PEC { ExternalAccessible := 'False'; ExternalVisible := 'False'; ExternalWritable := 'False'; S7_SetPoint := 'False'} : "UDT_PECStatus";   // PEC status structure
      ss_FIFOStatus { ExternalAccessible := 'False'; ExternalVisible := 'False'; ExternalWritable := 'False'; S7_SetPoint := 'False'} : "UDT_FifoStatus";   // Status structure
      s_R_TRIG_Connection {InstructionName := 'R_TRIG'; LibVersion := '1.0'; ExternalAccessible := 'False'; ExternalVisible := 'False'; ExternalWritable := 'False'; S7_SetPoint := 'False'} : R_TRIG;   // Rising edge trigger connection reastablished
      s_F_TRIG_SendAllErrors {InstructionName := 'F_TRIG'; LibVersion := '1.0'; ExternalAccessible := 'False'; ExternalVisible := 'False'; ExternalWritable := 'False'; S7_SetPoint := 'False'} : F_TRIG;   // Falling edge trigger from signal send all errors
      sdi_Code { ExternalAccessible := 'False'; ExternalVisible := 'False'; ExternalWritable := 'False'} : DInt;   // Error code
      si_State { ExternalAccessible := 'False'; ExternalVisible := 'False'; ExternalWritable := 'False'} : Int;   // Error state
      sx_ItemErrorMessageReq { ExternalAccessible := 'False'; ExternalVisible := 'False'; ExternalWritable := 'False'} : Bool;   // Item error message required
      sx_ItemErrorBlockError { ExternalAccessible := 'False'; ExternalVisible := 'False'; ExternalWritable := 'False'} : Bool;   // Item error block error
      sx_ItemErrorBlockWarning { ExternalAccessible := 'False'; ExternalVisible := 'False'; ExternalWritable := 'False'} : Bool;   // Item error block warning
      sx_SendAllProcedure { ExternalAccessible := 'False'; ExternalVisible := 'False'; ExternalWritable := 'False'} : Bool;   // Send all procedure
      sx_FIFOError { ExternalAccessible := 'False'; ExternalVisible := 'False'; ExternalWritable := 'False'} : Bool;   // FIFO Error
      sx_FIFOWarning { ExternalAccessible := 'False'; ExternalVisible := 'False'; ExternalWritable := 'False'} : Bool;   // FIFO Warning
   END_VAR

   VAR CONSTANT
      ci_MessageGroup : Int := 1;
      ci_TimeSpan : Int := 0;
   END_VAR


BEGIN
	(*
	----------------------------------------------------------------------------------------
	|                                                                                      |
	|  Copyright  2023             FORTNA Europe BV                                        |
	|  All Rights Reserved         Netherlands                                             |
	|                                                                                      |
	----------------------------------------------------------------------------------------
	Version history:
	Date        | Version   | Author       | Remark
	----------------------------------------------------------------------------------------
	03/01/2023  | 1.0       | S. Nikodem   | Release TIA 17 | DHL Munich 2023
	13/03/2023  | 1.1       | S. Nieswiec  | Updated for new Baseline
	*)

	REGION 1 - Initialize message required signals

	    #sx_ItemErrorMessageReq := FALSE;

	    // On connection re-establish send last remembered status and error state ( status only when it's diffrent then 0 )
	    #s_R_TRIG_Connection(CLK := #ix_MFCConnected);

	    IF #s_R_TRIG_Connection.Q
	    THEN
	        #sx_ItemErrorMessageReq := TRUE;
	    END_IF;

	    // Prepare trigger on the collective reset signal.
	    #s_F_TRIG_SendAllErrors(CLK := #ix_SendAllErrorsState);

	    // When collective reset will go down, start send every equipment errors.
	    IF #s_F_TRIG_SendAllErrors.Q AND NOT #sx_SendAllProcedure
	    THEN
	        #sx_SendAllProcedure := TRUE;
	    END_IF;

	END_REGION

	REGION 2 - FIFO header status update

	    // Mode 'S' - FIFO register status update.
	    "FC_Fifo"(ic_Mode := 'S',
	              qUDT_Status => #ss_FIFOStatus,
	              qx_Error => #sx_FIFOError,
	              qx_Warning => #sx_FIFOWarning,
	              iqv_Data := #s_UDT_Message,
	              iqUDT_FifoHeader := #iq_UDT_FifoHeader,
	              iqv_DataBuffer := #iqs_FifoData);

	END_REGION

	REGION 3 - Prepare message data

	    IF NOT #ix_CollectiveReset AND NOT #ss_FIFOStatus.FifoPreFull
	    THEN

	        //Copy input data to static memory
	        #s_UDT_PEC := #i_UDT_PECStatus;
	        // Check which specific status changed, prepare code, change state and write new status into the old one.

	        IF (#s_UDT_PEC.Jam <> #s_UDT_PECOLD.Jam)
	            OR (#sx_SendAllProcedure)
	            OR #sx_ItemErrorMessageReq
	        THEN
	            #sx_ItemErrorMessageReq := TRUE;
	            #sdi_Code := "DB_MFC_ErrorCode".PEC.Jam;
	            #si_State := BOOL_TO_INT(#s_UDT_PEC.Jam);
	            #s_UDT_PECOLD.Jam := #s_UDT_PEC.Jam;
	            #sx_SendAllProcedure := FALSE;
	        END_IF;

	        //The ELSIF needs to be tested
	    ELSIF #sx_ItemErrorMessageReq THEN
	        #sx_ItemErrorMessageReq := FALSE;
	    END_IF;


	END_REGION

	REGION 4 - Write message components to the item error structure

	    #s_UDT_ItemError.ItemNumber := #i_UDT_EquipmentNumber;
	    #s_UDT_ItemError.Error := #sdi_Code;
	    #s_UDT_ItemError.State := #si_State;
	    #s_UDT_ItemError.Masked := 1;

	END_REGION

	REGION 5 - Prepare messages to the MFC

	    // If item error message required signal is set, prepare the item error message.
	    IF (#sx_ItemErrorMessageReq)
	    THEN
	        #s_FB_ItemError(i_UDT_ItemErrorBody := #s_UDT_ItemError,
	                        ii_MessageGroup := #ci_MessageGroup,
	                        ix_FlagRetry := FALSE,
	                        idi_TimeSpan := #ci_TimeSpan,
	                        qx_Error => #sx_ItemErrorBlockError,
	                        qx_Warning => #sx_ItemErrorBlockWarning,
	                        iq_UDT_FifoHeader := #iq_UDT_FifoHeader,
	                        iqs_FifoData := #iqs_FifoData,
	                        iqdi_MessageSequenceNumber := #iqdi_MessageSequenceNumber);
	    END_IF;

	END_REGION

	REGION 6 - Write outputs

	    // Prepare collective output error.
	    #qx_Error := #sx_ItemErrorBlockError
	    OR #sx_FIFOError;

	    // Prepare collective output warning.
	    #qx_Warning := #sx_ItemErrorBlockWarning
	    OR #sx_FIFOWarning;

	END_REGION
END_FUNCTION_BLOCK

FUNCTION_BLOCK "FB_MFC_Visu_Heartbeat"
{ S7_Optimized_Access := 'TRUE' }
VERSION : 0.1
// ATTRIBUTES
// AUTO_NUMBER = True
// BLOCK_NUMBER = 150
// END_ATTRIBUTES
   VAR_INPUT
      iudi_HeartbeatInterval { ExternalAccessible := 'False'; ExternalVisible := 'False'; ExternalWritable := 'False'} : UDInt;   // Heartbeat send time interval [ms]
      ii_MessageGroup { ExternalAccessible := 'False'; ExternalVisible := 'False'; ExternalWritable := 'False'} : Int;   // Message group
      ix_FlagRetry { ExternalAccessible := 'False'; ExternalVisible := 'False'; ExternalWritable := 'False'} : Bool;   // TRUE when message is sent again
      idi_TimeSpan { ExternalAccessible := 'False'; ExternalVisible := 'False'; ExternalWritable := 'False'} : DInt;   // Time difference between messages
   END_VAR

   VAR_OUTPUT
      qx_Error { ExternalAccessible := 'False'; ExternalVisible := 'False'; ExternalWritable := 'False'} : Bool;   // TRUE when collective block error occurred
      qx_Warning { ExternalAccessible := 'False'; ExternalVisible := 'False'; ExternalWritable := 'False'} : Bool;   // TRUE when collective block warning occurred
   END_VAR

   VAR_IN_OUT
      iq_UDT_FifoHeader : "UDT_FifoHeader";   // FIFO header
      iqs_FifoData : Array[*] of "UDT_MessageV2";   // FIFO data buffer
      iqdi_MessageSequenceNumber { ExternalAccessible := 'False'; ExternalVisible := 'False'; ExternalWritable := 'False'} : DInt;   // Message number
   END_VAR

